LIN {X 0,Y 353.94,Z 241.157,A -85,B 0,C 180,E1 -13393.452,E2 -13393.452} C_VEL
LIN {X 0,Y 355.992,Z 254.031,A -85,B 0,C 180,E1 -13394.17,E2 -13394.17} C_VEL
LIN {X 0,Y 356.994,Z 264.311,A -85,B 0,C 180,E1 -13394.928,E2 -13394.928} C_VEL
LIN {X 0,Y 357.262,Z 272.08,A -85,B 0,C 180,E1 -13395.62,E2 -13395.62} C_VEL
LIN {X 0,Y 356.698,Z 280.213,A -85,B 0,C 180,E1 -13396.469,E2 -13396.469} C_VEL
LIN {X 0,Y 355.831,Z 287.972,A -85,B 0,C 180,E1 -13397.452,E2 -13397.452} C_VEL
LIN {X 0,Y 355.018,Z 296.94,A -85,B 0,C 180,E1 -13398.872,E2 -13398.872} C_VEL
LIN {X 0,Y 354.362,Z 303.882,A -85,B 0,C 180,E1 -13400.295,E2 -13400.295} C_VEL
LIN {X 0,Y 353.942,Z 308.46,A -85,B 0,C 180,E1 -13401.436,E2 -13401.436} C_VEL
LIN {X 0,Y 353.645,Z 312.278,A -85,B 0,C 180,E1 -13402.578,E2 -13402.578} C_VEL
LIN {X 0,Y 353.331,Z 316.635,A -85,B 0,C 180,E1 -13404.293,E2 -13404.293} C_VEL
LIN {X 0,Y 353.333,Z 318.872,A -85,B 0,C 180,E1 -13405.437,E2 -13405.437} C_VEL
LIN {X 0,Y 353.267,Z 320.538,A -85,B 0,C 180,E1 -13406.579,E2 -13406.579} C_VEL
LIN {X 0,Y 353.258,Z 321.597,A -85,B 0,C 180,E1 -13407.72,E2 -13407.72} C_VEL
LIN {X 0,Y 353.356,Z 322.159,A -85,B 0,C 180,E1 -13408.861,E2 -13408.861} C_VEL
LIN {X 0,Y 353.398,Z 322.239,A -85,B 0,C 180,E1 -13410,E2 -13410} C_VEL
LIN {X 0,Y 353.391,Z 321.836,A -85,B 0,C 180,E1 -13411.14,E2 -13411.14} C_VEL
LIN {X 0,Y 353.284,Z 320.881,A -85,B 0,C 180,E1 -13412.28,E2 -13412.28} C_VEL
LIN {X 0,Y 353.338,Z 318.39,A -85,B 0,C 180,E1 -13413.992,E2 -13413.992} C_VEL
LIN {X 0,Y 353.347,Z 316.056,A -85,B 0,C 180,E1 -13415.135,E2 -13415.135} C_VEL
LIN {X 0,Y 353.522,Z 311.248,A -85,B 0,C 180,E1 -13416.851,E2 -13416.851} C_VEL
LIN {X 0,Y 353.776,Z 306.025,A -85,B 0,C 180,E1 -13418.281,E2 -13418.281} C_VEL
LIN {X 0,Y 354.128,Z 300.895,A -85,B 0,C 180,E1 -13419.424,E2 -13419.424} C_VEL
LIN {X 0,Y 354.525,Z 294.697,A -85,B 0,C 180,E1 -13420.566,E2 -13420.566} C_VEL
LIN {X 0,Y 354.963,Z 288.171,A -85,B 0,C 180,E1 -13421.565,E2 -13421.565} C_VEL
LIN {X 0,Y 355.624,Z 280.281,A -85,B 0,C 180,E1 -13422.556,E2 -13422.556} C_VEL
LIN {X 0,Y 356.12,Z 271.928,A -85,B 0,C 180,E1 -13423.408,E2 -13423.408} C_VEL
LIN {X 0,Y 355.694,Z 262.322,A -85,B 0,C 180,E1 -13424.209,E2 -13424.209} C_VEL
LIN {X 0,Y 354.598,Z 250.562,A -85,B 0,C 180,E1 -13424.931,E2 -13424.931} C_VEL
LIN {X 0,Y 353.691,Z 242.124,A -85,B 0,C 180,E1 -13425.339,E2 -13425.339} C_VEL
LIN {X 0,Y 354.181,Z 233.988,A -85,B 0,C 180,E1 -13429.112,E2 -13429.112} C_VEL
LIN {X 0,Y 354.734,Z 226.313,A -85,B 0,C 180,E1 -13432.727,E2 -13432.727} C_VEL
LIN {X 0,Y 355.482,Z 218.591,A -85,B 0,C 180,E1 -13436.413,E2 -13436.413} C_VEL
LIN {X 0,Y 356.416,Z 210.762,A -85,B 0,C 180,E1 -13440.247,E2 -13440.247} C_VEL
LIN {X 0,Y 356.568,Z 207.213,A -85,B 0,C 180,E1 -13442.055,E2 -13442.055} C_VEL
LIN {X 0,Y 355.731,Z 201.801,A -85,B 0,C 180,E1 -13444.956,E2 -13444.956} C_VEL
LIN {X 0,Y 354.893,Z 197.094,A -85,B 0,C 180,E1 -13447.615,E2 -13447.615} C_VEL
LIN {X 0,Y 354.791,Z 197.102,A -85,B 0,C 180,E1 -13451.171,E2 -13451.171} C_VEL
LIN {X 0,Y 354.767,Z 197.108,A -85,B 0,C 180,E1 -13454.506,E2 -13454.506} C_VEL
LIN {X 0,Y 354.794,Z 197.101,A -85,B 0,C 180,E1 -13457.662,E2 -13457.662} C_VEL
LIN {X 0,Y 354.789,Z 197.103,A -85,B 0,C 180,E1 -13460.662,E2 -13460.662} C_VEL
LIN {X 0,Y 354.826,Z 197.101,A -85,B 0,C 180,E1 -13464.301,E2 -13464.301} C_VEL
LIN {X 0,Y 354.791,Z 197.103,A -85,B 0,C 180,E1 -13467.666,E2 -13467.666} C_VEL
LIN {X 0,Y 354.851,Z 197.096,A -85,B 0,C 180,E1 -13471.618,E2 -13471.618} C_VEL
LIN {X 0,Y 354.903,Z 197.09,A -85,B 0,C 180,E1 -13474.172,E2 -13474.172} C_VEL
LIN {X 0,Y 354.82,Z 197.102,A -85,B 0,C 180,E1 -13477.892,E2 -13477.892} C_VEL
LIN {X 0,Y 354.927,Z 197.088,A -85,B 0,C 180,E1 -13481.891,E2 -13481.891} C_VEL
LIN {X 0,Y 354.947,Z 197.083,A -85,B 0,C 180,E1 -13485.98,E2 -13485.98} C_VEL
LIN {X 0,Y 354.96,Z 197.083,A -85,B 0,C 180,E1 -13489.734,E2 -13489.734} C_VEL
LIN {X 0,Y 355.115,Z 197.065,A -85,B 0,C 180,E1 -13493.179,E2 -13493.179} C_VEL
LIN {X 0,Y 355.246,Z 197.046,A -85,B 0,C 180,E1 -13497.731,E2 -13497.731} C_VEL
LIN {X 0,Y 355.377,Z 197.028,A -85,B 0,C 180,E1 -13499.999,E2 -13499.999} C_VEL
LIN {X 0,Y 355.247,Z 197.044,A -85,B 0,C 180,E1 -13502.267,E2 -13502.267} C_VEL
LIN {X 0,Y 355.114,Z 197.065,A -85,B 0,C 180,E1 -13506.819,E2 -13506.819} C_VEL
LIN {X 0,Y 354.958,Z 197.081,A -85,B 0,C 180,E1 -13510.264,E2 -13510.264} C_VEL
LIN {X 0,Y 354.944,Z 197.082,A -85,B 0,C 180,E1 -13514.018,E2 -13514.018} C_VEL
LIN {X 0,Y 354.89,Z 197.089,A -85,B 0,C 180,E1 -13518.091,E2 -13518.091} C_VEL
LIN {X 0,Y 354.816,Z 197.1,A -85,B 0,C 180,E1 -13522.106,E2 -13522.106} C_VEL
LIN {X 0,Y 354.898,Z 197.088,A -85,B 0,C 180,E1 -13525.826,E2 -13525.826} C_VEL
LIN {X 0,Y 354.852,Z 197.094,A -85,B 0,C 180,E1 -13529.677,E2 -13529.677} C_VEL
LIN {X 0,Y 354.804,Z 197.101,A -85,B 0,C 180,E1 -13533.701,E2 -13533.701} C_VEL
LIN {X 0,Y 354.796,Z 197.104,A -85,B 0,C 180,E1 -13536.458,E2 -13536.458} C_VEL
LIN {X 0,Y 354.821,Z 197.097,A -85,B 0,C 180,E1 -13539.422,E2 -13539.422} C_VEL
LIN {X 0,Y 354.784,Z 197.102,A -85,B 0,C 180,E1 -13542.866,E2 -13542.866} C_VEL
LIN {X 0,Y 354.763,Z 197.108,A -85,B 0,C 180,E1 -13546.102,E2 -13546.102} C_VEL
LIN {X 0,Y 354.783,Z 197.103,A -85,B 0,C 180,E1 -13549.178,E2 -13549.178} C_VEL
LIN {X 0,Y 354.802,Z 197.1,A -85,B 0,C 180,E1 -13552.401,E2 -13552.401} C_VEL
LIN {X 0,Y 354.806,Z 197.099,A -85,B 0,C 180,E1 -13554.94,E2 -13554.94} C_VEL
LIN {X 0,Y 354.787,Z 197.102,A -85,B 0,C 180,E1 -13558.404,E2 -13558.404} C_VEL
LIN {X 0,Y 354.847,Z 197.098,A -85,B 0,C 180,E1 -13561.618,E2 -13561.618} C_VEL
LIN {X 0,Y 354.892,Z 197.089,A -85,B 0,C 180,E1 -13564.172,E2 -13564.172} C_VEL
LIN {X 0,Y 354.827,Z 197.098,A -85,B 0,C 180,E1 -13567.893,E2 -13567.893} C_VEL
LIN {X 0,Y 354.915,Z 197.086,A -85,B 0,C 180,E1 -13571.891,E2 -13571.891} C_VEL
LIN {X 0,Y 354.935,Z 197.083,A -85,B 0,C 180,E1 -13575.98,E2 -13575.98} C_VEL
LIN {X 0,Y 354.975,Z 197.078,A -85,B 0,C 180,E1 -13579.736,E2 -13579.736} C_VEL
LIN {X 0,Y 355.105,Z 197.062,A -85,B 0,C 180,E1 -13582.036,E2 -13582.036} C_VEL
LIN {X 0,Y 355.084,Z 197.065,A -85,B 0,C 180,E1 -13584.32,E2 -13584.32} C_VEL
LIN {X 0,Y 355.235,Z 197.045,A -85,B 0,C 180,E1 -13587.732,E2 -13587.732} C_VEL
LIN {X 0,Y 355.388,Z 197.027,A -85,B 0,C 180,E1 -13590,E2 -13590} C_VEL
LIN {X 0,Y 355.237,Z 197.047,A -85,B 0,C 180,E1 -13592.267,E2 -13592.267} C_VEL
LIN {X 0,Y 355.131,Z 197.062,A -85,B 0,C 180,E1 -13596.819,E2 -13596.819} C_VEL
LIN {X 0,Y 355.001,Z 197.076,A -85,B 0,C 180,E1 -13599.113,E2 -13599.113} C_VEL
LIN {X 0,Y 354.834,Z 197.1,A -85,B 0,C 180,E1 -13602.584,E2 -13602.584} C_VEL
LIN {X 0,Y 354.529,Z 197.156,A -85,B 0,C 180,E1 -13605.375,E2 -13605.375} C_VEL
LIN {X 0,Y 354.19,Z 201.044,A -85,B 0,C 180,E1 -13608.51,E2 -13608.51} C_VEL
LIN {X 0,Y 353.974,Z 205.678,A -85,B 0,C 180,E1 -13612.162,E2 -13612.162} C_VEL
LIN {X 0,Y 353.844,Z 208.876,A -85,B 0,C 180,E1 -13614.651,E2 -13614.651} C_VEL
LIN {X 0,Y 353.691,Z 212.209,A -85,B 0,C 180,E1 -13617.195,E2 -13617.195} C_VEL
LIN {X 0,Y 353.563,Z 216.799,A -85,B 0,C 180,E1 -13620.663,E2 -13620.663} C_VEL
LIN {X 0,Y 355.402,Z 227.901,A -85,B 0,C 180,E1 -13621.298,E2 -13621.298} C_VEL
LIN {X 0,Y 356.573,Z 235.778,A -85,B 0,C 180,E1 -13621.886,E2 -13621.886} C_VEL
LIN {X 0,Y 356.726,Z 240.779,A -85,B 0,C 180,E1 -13622.303,E2 -13622.303} C_VEL
LIN {X 0,Y 356.17,Z 249.655,A -85,B 0,C 180,E1 -13623.2,E2 -13623.2} C_VEL
LIN {X 0,Y 355.669,Z 257.094,A -85,B 0,C 180,E1 -13624.132,E2 -13624.132} C_VEL
LIN {X 0,Y 355.113,Z 264.014,A -85,B 0,C 180,E1 -13625.189,E2 -13625.189} C_VEL
LIN {X 0,Y 354.591,Z 270.903,A -85,B 0,C 180,E1 -13626.484,E2 -13626.484} C_VEL
LIN {X 0,Y 354.16,Z 277.029,A -85,B 0,C 180,E1 -13627.964,E2 -13627.964} C_VEL
LIN {X 0,Y 353.727,Z 281.835,A -85,B 0,C 180,E1 -13629.478,E2 -13629.478} C_VEL
LIN {X 0,Y 353.468,Z 285.305,A -85,B 0,C 180,E1 -13630.929,E2 -13630.929} C_VEL
LIN {X 0,Y 353.266,Z 288.109,A -85,B 0,C 180,E1 -13632.603,E2 -13632.603} C_VEL
LIN {X 0,Y 353.172,Z 289.652,A -85,B 0,C 180,E1 -13634.245,E2 -13634.245} C_VEL
LIN {X 0,Y 353.191,Z 290.008,A -85,B 0,C 180,E1 -13635.859,E2 -13635.859} C_VEL
LIN {X 0,Y 353.335,Z 289.319,A -85,B 0,C 180,E1 -13637.449,E2 -13637.449} C_VEL
LIN {X 0,Y 353.635,Z 287.419,A -85,B 0,C 180,E1 -13639.15,E2 -13639.15} C_VEL
LIN {X 0,Y 353.136,Z 285.956,A -85,B 0,C 180,E1 -13640.076,E2 -13640.076} C_VEL
LIN {X 0,Y 350.647,Z 283.004,A -85,B 0,C 180,E1 -13641.571,E2 -13641.571} C_VEL
LIN {X 0,Y 348.304,Z 279.171,A -85,B 0,C 180,E1 -13643.022,E2 -13643.022} C_VEL
LIN {X 0,Y 348.029,Z 276.23,A -85,B 0,C 180,E1 -13643.864,E2 -13643.864} C_VEL
LIN {X 0,Y 348.715,Z 270.077,A -85,B 0,C 180,E1 -13645.297,E2 -13645.297} C_VEL
LIN {X 0,Y 349.518,Z 263.05,A -85,B 0,C 180,E1 -13646.604,E2 -13646.604} C_VEL
LIN {X 0,Y 350.516,Z 254.114,A -85,B 0,C 180,E1 -13647.906,E2 -13647.906} C_VEL
LIN {X 0,Y 351.121,Z 246.314,A -85,B 0,C 180,E1 -13648.805,E2 -13648.805} C_VEL
LIN {X 0,Y 351.522,Z 241.461,A -85,B 0,C 180,E1 -13649.283,E2 -13649.283} C_VEL
LIN {X 0,Y 350.018,Z 231.844,A -85,B 0,C 180,E1 -13650.158,E2 -13650.158} C_VEL
LIN {X 0,Y 347.72,Z 221.982,A -85,B 0,C 180,E1 -13650.895,E2 -13650.895} C_VEL
LIN {X 0,Y 346.82,Z 218.272,A -85,B 0,C 180,E1 -13651.15,E2 -13651.15} C_VEL
LIN {X 0,Y 346.982,Z 215.406,A -85,B 0,C 180,E1 -13653.54,E2 -13653.54} C_VEL
LIN {X 0,Y 347.236,Z 210.883,A -85,B 0,C 180,E1 -13657.385,E2 -13657.385} C_VEL
LIN {X 0,Y 347.542,Z 206.631,A -85,B 0,C 180,E1 -13661.123,E2 -13661.123} C_VEL
LIN {X 0,Y 347.864,Z 202.634,A -85,B 0,C 180,E1 -13664.774,E2 -13664.774} C_VEL
LIN {X 0,Y 347.994,Z 200.093,A -85,B 0,C 180,E1 -13667.166,E2 -13667.166} C_VEL
LIN {X 0,Y 347.885,Z 197.966,A -85,B 0,C 180,E1 -13669.525,E2 -13669.525} C_VEL
LIN {X 0,Y 348.079,Z 197.946,A -85,B 0,C 180,E1 -13671.876,E2 -13671.876} C_VEL
LIN {X 0,Y 348.068,Z 197.949,A -85,B 0,C 180,E1 -13674.207,E2 -13674.207} C_VEL
LIN {X 0,Y 348.207,Z 197.926,A -85,B 0,C 180,E1 -13677.688,E2 -13677.688} C_VEL
LIN {X 0,Y 348.369,Z 197.905,A -85,B 0,C 180,E1 -13680.001,E2 -13680.001} C_VEL
LIN {X 0,Y 348.207,Z 197.926,A -85,B 0,C 180,E1 -13682.314,E2 -13682.314} C_VEL
LIN {X 0,Y 348.081,Z 197.942,A -85,B 0,C 180,E1 -13686.959,E2 -13686.959} C_VEL
LIN {X 0,Y 347.899,Z 197.963,A -85,B 0,C 180,E1 -13690.476,E2 -13690.476} C_VEL
LIN {X 0,Y 347.9,Z 197.963,A -85,B 0,C 180,E1 -13694.151,E2 -13694.151} C_VEL
LIN {X 0,Y 347.894,Z 197.964,A -85,B 0,C 180,E1 -13698.291,E2 -13698.291} C_VEL
LIN {X 0,Y 347.791,Z 197.977,A -85,B 0,C 180,E1 -13701.636,E2 -13701.636} C_VEL
LIN {X 0,Y 347.814,Z 197.97,A -85,B 0,C 180,E1 -13705.109,E2 -13705.109} C_VEL
LIN {X 0,Y 347.812,Z 197.974,A -85,B 0,C 180,E1 -13707.695,E2 -13707.695} C_VEL
LIN {X 0,Y 347.766,Z 197.979,A -85,B 0,C 180,E1 -13710.347,E2 -13710.347} C_VEL
LIN {X 0,Y 347.746,Z 197.982,A -85,B 0,C 180,E1 -13714.464,E2 -13714.464} C_VEL
LIN {X 0,Y 347.775,Z 197.98,A -85,B 0,C 180,E1 -13717.989,E2 -13717.989} C_VEL
LIN {X 0,Y 347.753,Z 197.984,A -85,B 0,C 180,E1 -13721.831,E2 -13721.831} C_VEL
LIN {X 0,Y 347.708,Z 197.991,A -85,B 0,C 180,E1 -13725.027,E2 -13725.027} C_VEL
LIN {X 0,Y 347.79,Z 198.146,A -85,B 0,C 180,E1 -13728.948,E2 -13728.948} C_VEL
LIN {X 0,Y 348.556,Z 202.078,A -85,B 0,C 180,E1 -13731.848,E2 -13731.848} C_VEL
LIN {X 0,Y 349.657,Z 207.924,A -85,B 0,C 180,E1 -13735.751,E2 -13735.751} C_VEL
LIN {X 0,Y 350.09,Z 210.716,A -85,B 0,C 180,E1 -13737.475,E2 -13737.475} C_VEL
LIN {X 0,Y 349.935,Z 213.693,A -85,B 0,C 180,E1 -13739.195,E2 -13739.195} C_VEL
LIN {X 0,Y 348.847,Z 220.858,A -85,B 0,C 180,E1 -13743.045,E2 -13743.045} C_VEL
LIN {X 0,Y 347.96,Z 228.169,A -85,B 0,C 180,E1 -13746.806,E2 -13746.806} C_VEL
LIN {X 0,Y 347.292,Z 235.615,A -85,B 0,C 180,E1 -13750.494,E2 -13750.494} C_VEL
LIN {X 0,Y 346.929,Z 241.06,A -85,B 0,C 180,E1 -13753.051,E2 -13753.051} C_VEL
LIN {X 0,Y 349.037,Z 253.685,A -85,B 0,C 180,E1 -13753.777,E2 -13753.777} C_VEL
LIN {X 0,Y 350.037,Z 263.552,A -85,B 0,C 180,E1 -13754.525,E2 -13754.525} C_VEL
LIN {X 0,Y 350.341,Z 272.338,A -85,B 0,C 180,E1 -13755.329,E2 -13755.329} C_VEL
LIN {X 0,Y 349.815,Z 280.367,A -85,B 0,C 180,E1 -13756.198,E2 -13756.198} C_VEL
LIN {X 0,Y 348.917,Z 288.047,A -85,B 0,C 180,E1 -13757.199,E2 -13757.199} C_VEL
LIN {X 0,Y 348.057,Z 296.92,A -85,B 0,C 180,E1 -13758.646,E2 -13758.646} C_VEL
LIN {X 0,Y 347.339,Z 303.789,A -85,B 0,C 180,E1 -13760.097,E2 -13760.097} C_VEL
LIN {X 0,Y 346.903,Z 308.325,A -85,B 0,C 180,E1 -13761.261,E2 -13761.261} C_VEL
LIN {X 0,Y 346.572,Z 312.11,A -85,B 0,C 180,E1 -13762.426,E2 -13762.426} C_VEL
LIN {X 0,Y 346.251,Z 316.425,A -85,B 0,C 180,E1 -13764.175,E2 -13764.175} C_VEL
LIN {X 0,Y 346.245,Z 318.624,A -85,B 0,C 180,E1 -13765.343,E2 -13765.343} C_VEL
LIN {X 0,Y 346.189,Z 320.273,A -85,B 0,C 180,E1 -13766.509,E2 -13766.509} C_VEL
LIN {X 0,Y 346.164,Z 321.315,A -85,B 0,C 180,E1 -13767.673,E2 -13767.673} C_VEL
LIN {X 0,Y 346.257,Z 321.845,A -85,B 0,C 180,E1 -13768.837,E2 -13768.837} C_VEL
LIN {X 0,Y 346.318,Z 321.895,A -85,B 0,C 180,E1 -13770,E2 -13770} C_VEL
LIN {X 0,Y 346.294,Z 321.46,A -85,B 0,C 180,E1 -13771.163,E2 -13771.163} C_VEL
LIN {X 0,Y 346.188,Z 320.496,A -85,B 0,C 180,E1 -13772.327,E2 -13772.327} C_VEL
LIN {X 0,Y 346.269,Z 317.952,A -85,B 0,C 180,E1 -13774.074,E2 -13774.074} C_VEL
LIN {X 0,Y 346.246,Z 315.595,A -85,B 0,C 180,E1 -13775.241,E2 -13775.241} C_VEL
LIN {X 0,Y 346.444,Z 310.731,A -85,B 0,C 180,E1 -13776.991,E2 -13776.991} C_VEL
LIN {X 0,Y 346.741,Z 305.465,A -85,B 0,C 180,E1 -13778.45,E2 -13778.45} C_VEL
LIN {X 0,Y 347.065,Z 300.279,A -85,B 0,C 180,E1 -13779.617,E2 -13779.617} C_VEL
LIN {X 0,Y 347.534,Z 294.026,A -85,B 0,C 180,E1 -13780.781,E2 -13780.781} C_VEL
LIN {X 0,Y 348.111,Z 286.412,A -85,B 0,C 180,E1 -13781.943,E2 -13781.943} C_VEL
LIN {X 0,Y 348.889,Z 276.928,A -85,B 0,C 180,E1 -13783.098,E2 -13783.098} C_VEL
LIN {X 0,Y 349.088,Z 269.405,A -85,B 0,C 180,E1 -13783.832,E2 -13783.832} C_VEL
LIN {X 0,Y 348.361,Z 259.219,A -85,B 0,C 180,E1 -13784.63,E2 -13784.63} C_VEL
LIN {X 0,Y 347.423,Z 249.351,A -85,B 0,C 180,E1 -13785.218,E2 -13785.218} C_VEL
LIN {X 0,Y 346.638,Z 241.909,A -85,B 0,C 180,E1 -13785.584,E2 -13785.584} C_VEL
LIN {X 0,Y 347.139,Z 233.624,A -85,B 0,C 180,E1 -13789.515,E2 -13789.515} C_VEL
LIN {X 0,Y 347.646,Z 227.22,A -85,B 0,C 180,E1 -13792.588,E2 -13792.588} C_VEL
LIN {X 0,Y 348.397,Z 219.537,A -85,B 0,C 180,E1 -13796.346,E2 -13796.346} C_VEL
LIN {X 0,Y 349.352,Z 211.86,A -85,B 0,C 180,E1 -13800.194,E2 -13800.194} C_VEL
LIN {X 0,Y 349.616,Z 209.278,A -85,B 0,C 180,E1 -13801.511,E2 -13801.511} C_VEL
LIN {X 0,Y 348.935,Z 204.077,A -85,B 0,C 180,E1 -13804.33,E2 -13804.33} C_VEL
LIN {X 0,Y 347.841,Z 197.972,A -85,B 0,C 180,E1 -13807.899,E2 -13807.899} C_VEL
LIN {X 0,Y 347.754,Z 197.978,A -85,B 0,C 180,E1 -13811.83,E2 -13811.83} C_VEL
LIN {X 0,Y 347.709,Z 197.984,A -85,B 0,C 180,E1 -13815.027,E2 -13815.027} C_VEL
LIN {X 0,Y 347.751,Z 197.982,A -85,B 0,C 180,E1 -13818.398,E2 -13818.398} C_VEL
LIN {X 0,Y 347.768,Z 197.979,A -85,B 0,C 180,E1 -13822.013,E2 -13822.013} C_VEL
LIN {X 0,Y 347.749,Z 197.979,A -85,B 0,C 180,E1 -13825.536,E2 -13825.536} C_VEL
LIN {X 0,Y 347.749,Z 197.981,A -85,B 0,C 180,E1 -13828.3,E2 -13828.3} C_VEL
LIN {X 0,Y 347.783,Z 197.974,A -85,B 0,C 180,E1 -13830.987,E2 -13830.987} C_VEL
LIN {X 0,Y 347.835,Z 197.97,A -85,B 0,C 180,E1 -13833.607,E2 -13833.607} C_VEL
LIN {X 0,Y 347.789,Z 197.976,A -85,B 0,C 180,E1 -13836.161,E2 -13836.161} C_VEL
LIN {X 0,Y 347.813,Z 197.974,A -85,B 0,C 180,E1 -13839.909,E2 -13839.909} C_VEL
LIN {X 0,Y 347.871,Z 197.963,A -85,B 0,C 180,E1 -13842.359,E2 -13842.359} C_VEL
LIN {X 0,Y 347.902,Z 197.961,A -85,B 0,C 180,E1 -13845.97,E2 -13845.97} C_VEL
LIN {X 0,Y 347.901,Z 197.964,A -85,B 0,C 180,E1 -13849.524,E2 -13849.524} C_VEL
LIN {X 0,Y 348.081,Z 197.939,A -85,B 0,C 180,E1 -13853.041,E2 -13853.041} C_VEL
LIN {X 0,Y 348.209,Z 197.922,A -85,B 0,C 180,E1 -13857.686,E2 -13857.686} C_VEL
LIN {X 0,Y 348.327,Z 197.906,A -85,B 0,C 180,E1 -13859.999,E2 -13859.999} C_VEL
LIN {X 0,Y 348.209,Z 197.921,A -85,B 0,C 180,E1 -13862.312,E2 -13862.312} C_VEL
LIN {X 0,Y 348.08,Z 197.942,A -85,B 0,C 180,E1 -13866.957,E2 -13866.957} C_VEL
LIN {X 0,Y 347.899,Z 197.961,A -85,B 0,C 180,E1 -13870.474,E2 -13870.474} C_VEL
LIN {X 0,Y 347.9,Z 197.96,A -85,B 0,C 180,E1 -13874.149,E2 -13874.149} C_VEL
LIN {X 0,Y 347.829,Z 197.97,A -85,B 0,C 180,E1 -13878.258,E2 -13878.258} C_VEL
LIN {X 0,Y 347.767,Z 197.976,A -85,B 0,C 180,E1 -13881.625,E2 -13881.625} C_VEL
LIN {X 0,Y 347.81,Z 197.971,A -85,B 0,C 180,E1 -13885.107,E2 -13885.107} C_VEL
LIN {X 0,Y 347.81,Z 197.971,A -85,B 0,C 180,E1 -13887.692,E2 -13887.692} C_VEL
LIN {X 0,Y 347.762,Z 197.981,A -85,B 0,C 180,E1 -13890.345,E2 -13890.345} C_VEL
LIN {X 0,Y 347.742,Z 197.982,A -85,B 0,C 180,E1 -13894.463,E2 -13894.463} C_VEL
LIN {X 0,Y 347.771,Z 197.98,A -85,B 0,C 180,E1 -13897.987,E2 -13897.987} C_VEL
LIN {X 0,Y 347.747,Z 197.982,A -85,B 0,C 180,E1 -13901.829,E2 -13901.829} C_VEL
LIN {X 0,Y 347.701,Z 197.984,A -85,B 0,C 180,E1 -13905.026,E2 -13905.026} C_VEL
LIN {X 0,Y 347.745,Z 197.98,A -85,B 0,C 180,E1 -13908.396,E2 -13908.396} C_VEL
LIN {X 0,Y 347.769,Z 197.979,A -85,B 0,C 180,E1 -13912.01,E2 -13912.01} C_VEL
LIN {X 0,Y 347.738,Z 197.984,A -85,B 0,C 180,E1 -13915.535,E2 -13915.535} C_VEL
LIN {X 0,Y 347.758,Z 197.982,A -85,B 0,C 180,E1 -13919.653,E2 -13919.653} C_VEL
LIN {X 0,Y 347.846,Z 197.966,A -85,B 0,C 180,E1 -13922.743,E2 -13922.743} C_VEL
LIN {X 0,Y 347.781,Z 197.974,A -85,B 0,C 180,E1 -13926.161,E2 -13926.161} C_VEL
LIN {X 0,Y 347.81,Z 197.971,A -85,B 0,C 180,E1 -13929.909,E2 -13929.909} C_VEL
LIN {X 0,Y 347.859,Z 197.964,A -85,B 0,C 180,E1 -13932.359,E2 -13932.359} C_VEL
LIN {X 0,Y 347.889,Z 197.96,A -85,B 0,C 180,E1 -13935.97,E2 -13935.97} C_VEL
LIN {X 0,Y 347.925,Z 197.957,A -85,B 0,C 180,E1 -13939.525,E2 -13939.525} C_VEL
LIN {X 0,Y 348.066,Z 197.939,A -85,B 0,C 180,E1 -13941.874,E2 -13941.874} C_VEL
LIN {X 0,Y 348.059,Z 197.94,A -85,B 0,C 180,E1 -13944.205,E2 -13944.205} C_VEL
LIN {X 0,Y 348.197,Z 197.922,A -85,B 0,C 180,E1 -13947.686,E2 -13947.686} C_VEL
LIN {X 0,Y 348.337,Z 197.905,A -85,B 0,C 180,E1 -13950,E2 -13950} C_VEL
LIN {X 0,Y 348.199,Z 197.924,A -85,B 0,C 180,E1 -13952.313,E2 -13952.313} C_VEL
LIN {X 0,Y 348.099,Z 197.937,A -85,B 0,C 180,E1 -13956.958,E2 -13956.958} C_VEL
LIN {X 0,Y 347.936,Z 197.955,A -85,B 0,C 180,E1 -13959.299,E2 -13959.299} C_VEL
LIN {X 0,Y 347.79,Z 197.975,A -85,B 0,C 180,E1 -13962.843,E2 -13962.843} C_VEL
LIN {X 0,Y 347.442,Z 198.211,A -85,B 0,C 180,E1 -13965.546,E2 -13965.546} C_VEL
LIN {X 0,Y 347.112,Z 202.33,A -85,B 0,C 180,E1 -13968.902,E2 -13968.902} C_VEL
LIN {X 0,Y 346.975,Z 205.423,A -85,B 0,C 180,E1 -13971.382,E2 -13971.382} C_VEL
LIN {X 0,Y 346.746,Z 210.268,A -85,B 0,C 180,E1 -13975.191,E2 -13975.191} C_VEL
LIN {X 0,Y 346.575,Z 213.619,A -85,B 0,C 180,E1 -13977.801,E2 -13977.801} C_VEL
LIN {X 0,Y 346.505,Z 217.067,A -85,B 0,C 180,E1 -13980.424,E2 -13980.424} C_VEL
LIN {X 0,Y 348.301,Z 227.835,A -85,B 0,C 180,E1 -13981.051,E2 -13981.051} C_VEL
LIN {X 0,Y 349.549,Z 236.356,A -85,B 0,C 180,E1 -13981.7,E2 -13981.7} C_VEL
LIN {X 0,Y 349.73,Z 241.206,A -85,B 0,C 180,E1 -13982.116,E2 -13982.116} C_VEL
LIN {X 0,Y 349.122,Z 250.603,A -85,B 0,C 180,E1 -13983.096,E2 -13983.096} C_VEL
LIN {X 0,Y 348.578,Z 258.652,A -85,B 0,C 180,E1 -13984.148,E2 -13984.148} C_VEL
LIN {X 0,Y 347.867,Z 266.954,A -85,B 0,C 180,E1 -13985.509,E2 -13985.509} C_VEL
LIN {X 0,Y 347.357,Z 273.993,A -85,B 0,C 180,E1 -13987.023,E2 -13987.023} C_VEL
LIN {X 0,Y 346.934,Z 278.896,A -85,B 0,C 180,E1 -13988.344,E2 -13988.344} C_VEL
LIN {X 0,Y 346.599,Z 282.619,A -85,B 0,C 180,E1 -13989.601,E2 -13989.601} C_VEL
LIN {X 0,Y 346.326,Z 286.508,A -85,B 0,C 180,E1 -13991.339,E2 -13991.339} C_VEL
LIN {X 0,Y 346.13,Z 288.929,A -85,B 0,C 180,E1 -13993.035,E2 -13993.035} C_VEL
LIN {X 0,Y 346.066,Z 290.317,A -85,B 0,C 180,E1 -13995.299,E2 -13995.299} C_VEL
LIN {X 0,Y 346.177,Z 290.088,A -85,B 0,C 180,E1 -13996.959,E2 -13996.959} C_VEL
LIN {X 0,Y 346.452,Z 288.663,A -85,B 0,C 180,E1 -13998.64,E2 -13998.64} C_VEL
LIN {X 0,Y 346.806,Z 285.979,A -85,B 0,C 180,E1 -14000.36,E2 -14000.36} C_VEL
LIN {X 0,Y 347.161,Z 283.128,A -85,B 0,C 180,E1 -14001.648,E2 -14001.648} C_VEL
LIN {X 0,Y 347.788,Z 278.206,A -85,B 0,C 180,E1 -14003.315,E2 -14003.315} C_VEL
LIN {X 0,Y 348.029,Z 276.23,A -85,B 0,C 180,E1 -14003.864,E2 -14003.864} C_VEL
LIN {X 0,Y 347.773,Z 273.111,A -85,B 0,C 180,E1 -14004.676,E2 -14004.676} C_VEL
LIN {X 0,Y 345.608,Z 267.605,A -85,B 0,C 180,E1 -14005.986,E2 -14005.986} C_VEL
LIN {X 0,Y 343.539,Z 261.333,A -85,B 0,C 180,E1 -14007.228,E2 -14007.228} C_VEL
LIN {X 0,Y 343.409,Z 256.965,A -85,B 0,C 180,E1 -14007.905,E2 -14007.905} C_VEL
LIN {X 0,Y 344.348,Z 246.796,A -85,B 0,C 180,E1 -14009.147,E2 -14009.147} C_VEL
LIN {X 0,Y 344.711,Z 242.533,A -85,B 0,C 180,E1 -14009.578,E2 -14009.578} C_VEL
LIN {X 0,Y 343.087,Z 232.251,A -85,B 0,C 180,E1 -14010.554,E2 -14010.554} C_VEL
LIN {X 0,Y 340.653,Z 222.105,A -85,B 0,C 180,E1 -14011.338,E2 -14011.338} C_VEL
LIN {X 0,Y 339.8,Z 218.575,A -85,B 0,C 180,E1 -14011.596,E2 -14011.596} C_VEL
LIN {X 0,Y 340.036,Z 213.92,A -85,B 0,C 180,E1 -14015.585,E2 -14015.585} C_VEL
LIN {X 0,Y 340.354,Z 209.546,A -85,B 0,C 180,E1 -14019.451,E2 -14019.451} C_VEL
LIN {X 0,Y 340.648,Z 206.74,A -85,B 0,C 180,E1 -14021.974,E2 -14021.974} C_VEL
LIN {X 0,Y 340.949,Z 202.812,A -85,B 0,C 180,E1 -14025.68,E2 -14025.68} C_VEL
LIN {X 0,Y 340.955,Z 200.362,A -85,B 0,C 180,E1 -14028.106,E2 -14028.106} C_VEL
LIN {X 0,Y 340.893,Z 199.19,A -85,B 0,C 180,E1 -14029.308,E2 -14029.308} C_VEL
LIN {X 0,Y 341.043,Z 198.822,A -85,B 0,C 180,E1 -14031.707,E2 -14031.707} C_VEL
LIN {X 0,Y 341.044,Z 198.825,A -85,B 0,C 180,E1 -14034.087,E2 -14034.087} C_VEL
LIN {X 0,Y 341.169,Z 198.803,A -85,B 0,C 180,E1 -14037.64,E2 -14037.64} C_VEL
LIN {X 0,Y 341.317,Z 198.783,A -85,B 0,C 180,E1 -14040.001,E2 -14040.001} C_VEL
LIN {X 0,Y 341.169,Z 198.803,A -85,B 0,C 180,E1 -14042.362,E2 -14042.362} C_VEL
LIN {X 0,Y 341.049,Z 198.817,A -85,B 0,C 180,E1 -14047.103,E2 -14047.103} C_VEL
LIN {X 0,Y 340.85,Z 198.842,A -85,B 0,C 180,E1 -14050.695,E2 -14050.695} C_VEL
LIN {X 0,Y 340.865,Z 198.838,A -85,B 0,C 180,E1 -14054.326,E2 -14054.326} C_VEL
LIN {X 0,Y 340.84,Z 198.843,A -85,B 0,C 180,E1 -14058.468,E2 -14058.468} C_VEL
LIN {X 0,Y 340.756,Z 198.853,A -85,B 0,C 180,E1 -14061.858,E2 -14061.858} C_VEL
LIN {X 0,Y 340.775,Z 198.846,A -85,B 0,C 180,E1 -14065.665,E2 -14065.665} C_VEL
LIN {X 0,Y 340.742,Z 198.855,A -85,B 0,C 180,E1 -14068.32,E2 -14068.32} C_VEL
LIN {X 0,Y 340.706,Z 198.859,A -85,B 0,C 180,E1 -14071.045,E2 -14071.045} C_VEL
LIN {X 0,Y 340.72,Z 198.856,A -85,B 0,C 180,E1 -14075.279,E2 -14075.279} C_VEL
LIN {X 0,Y 340.712,Z 198.859,A -85,B 0,C 180,E1 -14078.386,E2 -14078.386} C_VEL
LIN {X 0,Y 340.701,Z 198.863,A -85,B 0,C 180,E1 -14082.046,E2 -14082.046} C_VEL
LIN {X 0,Y 340.654,Z 198.869,A -85,B 0,C 180,E1 -14086.227,E2 -14086.227} C_VEL
LIN {X 0,Y 340.731,Z 198.987,A -85,B 0,C 180,E1 -14088.329,E2 -14088.329} C_VEL
LIN {X 0,Y 341.634,Z 203.675,A -85,B 0,C 180,E1 -14091.892,E2 -14091.892} C_VEL
LIN {X 0,Y 342.507,Z 208.437,A -85,B 0,C 180,E1 -14095.163,E2 -14095.163} C_VEL
LIN {X 0,Y 343.103,Z 212.604,A -85,B 0,C 180,E1 -14097.821,E2 -14097.821} C_VEL
LIN {X 0,Y 342.859,Z 215.359,A -85,B 0,C 180,E1 -14099.422,E2 -14099.422} C_VEL
LIN {X 0,Y 341.787,Z 222.053,A -85,B 0,C 180,E1 -14103.104,E2 -14103.104} C_VEL
LIN {X 0,Y 341.01,Z 228.107,A -85,B 0,C 180,E1 -14106.304,E2 -14106.304} C_VEL
LIN {X 0,Y 340.285,Z 235.513,A -85,B 0,C 180,E1 -14110.076,E2 -14110.076} C_VEL
LIN {X 0,Y 339.917,Z 240.583,A -85,B 0,C 180,E1 -14112.594,E2 -14112.594} C_VEL
LIN {X 0,Y 342.074,Z 253.386,A -85,B 0,C 180,E1 -14113.361,E2 -14113.361} C_VEL
LIN {X 0,Y 343.094,Z 263.082,A -85,B 0,C 180,E1 -14114.115,E2 -14114.115} C_VEL
LIN {X 0,Y 343.444,Z 271.242,A -85,B 0,C 180,E1 -14114.876,E2 -14114.876} C_VEL
LIN {X 0,Y 343.07,Z 279.368,A -85,B 0,C 180,E1 -14115.769,E2 -14115.769} C_VEL
LIN {X 0,Y 342.154,Z 287.139,A -85,B 0,C 180,E1 -14116.791,E2 -14116.791} C_VEL
LIN {X 0,Y 341.464,Z 293.586,A -85,B 0,C 180,E1 -14117.821,E2 -14117.821} C_VEL
LIN {X 0,Y 340.751,Z 299.75,A -85,B 0,C 180,E1 -14119.002,E2 -14119.002} C_VEL
LIN {X 0,Y 340.081,Z 306.072,A -85,B 0,C 180,E1 -14120.484,E2 -14120.484} C_VEL
LIN {X 0,Y 339.527,Z 311.937,A -85,B 0,C 180,E1 -14122.268,E2 -14122.268} C_VEL
LIN {X 0,Y 339.256,Z 315.007,A -85,B 0,C 180,E1 -14123.458,E2 -14123.458} C_VEL
LIN {X 0,Y 339.139,Z 318.378,A -85,B 0,C 180,E1 -14125.245,E2 -14125.245} C_VEL
LIN {X 0,Y 339.114,Z 320.008,A -85,B 0,C 180,E1 -14126.436,E2 -14126.436} C_VEL
LIN {X 0,Y 339.074,Z 321.038,A -85,B 0,C 180,E1 -14127.624,E2 -14127.624} C_VEL
LIN {X 0,Y 339.159,Z 321.532,A -85,B 0,C 180,E1 -14128.813,E2 -14128.813} C_VEL
LIN {X 0,Y 339.226,Z 321.546,A -85,B 0,C 180,E1 -14130,E2 -14130} C_VEL
LIN {X 0,Y 339.197,Z 321.074,A -85,B 0,C 180,E1 -14131.187,E2 -14131.187} C_VEL
LIN {X 0,Y 339.097,Z 320.09,A -85,B 0,C 180,E1 -14132.376,E2 -14132.376} C_VEL
LIN {X 0,Y 339.2,Z 317.488,A -85,B 0,C 180,E1 -14134.159,E2 -14134.159} C_VEL
LIN {X 0,Y 339.209,Z 313.422,A -85,B 0,C 180,E1 -14136.007,E2 -14136.007} C_VEL
LIN {X 0,Y 339.506,Z 308.253,A -85,B 0,C 180,E1 -14137.733,E2 -14137.733} C_VEL
LIN {X 0,Y 339.96,Z 301.029,A -85,B 0,C 180,E1 -14139.52,E2 -14139.52} C_VEL
LIN {X 0,Y 340.402,Z 294.985,A -85,B 0,C 180,E1 -14140.709,E2 -14140.709} C_VEL
LIN {X 0,Y 340.92,Z 287.614,A -85,B 0,C 180,E1 -14141.897,E2 -14141.897} C_VEL
LIN {X 0,Y 341.632,Z 279.739,A -85,B 0,C 180,E1 -14142.928,E2 -14142.928} C_VEL
LIN {X 0,Y 342.107,Z 271.393,A -85,B 0,C 180,E1 -14143.817,E2 -14143.817} C_VEL
LIN {X 0,Y 341.503,Z 261.169,A -85,B 0,C 180,E1 -14144.704,E2 -14144.704} C_VEL
LIN {X 0,Y 340.406,Z 249.59,A -85,B 0,C 180,E1 -14145.432,E2 -14145.432} C_VEL
LIN {X 0,Y 339.577,Z 241.639,A -85,B 0,C 180,E1 -14145.839,E2 -14145.839} C_VEL
LIN {X 0,Y 340.024,Z 234.507,A -85,B 0,C 180,E1 -14149.312,E2 -14149.312} C_VEL
LIN {X 0,Y 340.646,Z 226.868,A -85,B 0,C 180,E1 -14153.079,E2 -14153.079} C_VEL
LIN {X 0,Y 341.469,Z 219.201,A -85,B 0,C 180,E1 -14156.924,E2 -14156.924} C_VEL
LIN {X 0,Y 342.474,Z 211.518,A -85,B 0,C 180,E1 -14160.866,E2 -14160.866} C_VEL
LIN {X 0,Y 342.392,Z 208.123,A -85,B 0,C 180,E1 -14162.693,E2 -14162.693} C_VEL
LIN {X 0,Y 341.417,Z 202.537,A -85,B 0,C 180,E1 -14165.857,E2 -14165.857} C_VEL
LIN {X 0,Y 340.791,Z 198.85,A -85,B 0,C 180,E1 -14168.032,E2 -14168.032} C_VEL
LIN {X 0,Y 340.703,Z 198.857,A -85,B 0,C 180,E1 -14172.045,E2 -14172.045} C_VEL
LIN {X 0,Y 340.655,Z 198.866,A -85,B 0,C 180,E1 -14176.227,E2 -14176.227} C_VEL
LIN {X 0,Y 340.678,Z 198.86,A -85,B 0,C 180,E1 -14179.756,E2 -14179.756} C_VEL
LIN {X 0,Y 340.707,Z 198.855,A -85,B 0,C 180,E1 -14183.258,E2 -14183.258} C_VEL
LIN {X 0,Y 340.697,Z 198.861,A -85,B 0,C 180,E1 -14186.153,E2 -14186.153} C_VEL
LIN {X 0,Y 340.746,Z 198.853,A -85,B 0,C 180,E1 -14190.329,E2 -14190.329} C_VEL
LIN {X 0,Y 340.808,Z 198.842,A -85,B 0,C 180,E1 -14193.019,E2 -14193.019} C_VEL
LIN {X 0,Y 340.759,Z 198.852,A -85,B 0,C 180,E1 -14195.638,E2 -14195.638} C_VEL
LIN {X 0,Y 340.74,Z 198.854,A -85,B 0,C 180,E1 -14199.473,E2 -14199.473} C_VEL
LIN {X 0,Y 340.862,Z 198.838,A -85,B 0,C 180,E1 -14201.984,E2 -14201.984} C_VEL
LIN {X 0,Y 340.874,Z 198.839,A -85,B 0,C 180,E1 -14205.704,E2 -14205.704} C_VEL
LIN {X 0,Y 340.852,Z 198.841,A -85,B 0,C 180,E1 -14209.305,E2 -14209.305} C_VEL
LIN {X 0,Y 341.049,Z 198.814,A -85,B 0,C 180,E1 -14212.897,E2 -14212.897} C_VEL
LIN {X 0,Y 341.17,Z 198.799,A -85,B 0,C 180,E1 -14217.638,E2 -14217.638} C_VEL
LIN {X 0,Y 341.278,Z 198.784,A -85,B 0,C 180,E1 -14219.999,E2 -14219.999} C_VEL
LIN {X 0,Y 341.171,Z 198.797,A -85,B 0,C 180,E1 -14222.36,E2 -14222.36} C_VEL
LIN {X 0,Y 341.048,Z 198.817,A -85,B 0,C 180,E1 -14227.101,E2 -14227.101} C_VEL
LIN {X 0,Y 340.85,Z 198.841,A -85,B 0,C 180,E1 -14230.693,E2 -14230.693} C_VEL
LIN {X 0,Y 340.864,Z 198.837,A -85,B 0,C 180,E1 -14234.324,E2 -14234.324} C_VEL
LIN {X 0,Y 340.786,Z 198.849,A -85,B 0,C 180,E1 -14238.439,E2 -14238.439} C_VEL
LIN {X 0,Y 340.717,Z 198.854,A -85,B 0,C 180,E1 -14241.84,E2 -14241.84} C_VEL
LIN {X 0,Y 340.772,Z 198.847,A -85,B 0,C 180,E1 -14245.663,E2 -14245.663} C_VEL
LIN {X 0,Y 340.74,Z 198.856,A -85,B 0,C 180,E1 -14248.318,E2 -14248.318} C_VEL
LIN {X 0,Y 340.702,Z 198.856,A -85,B 0,C 180,E1 -14251.043,E2 -14251.043} C_VEL
LIN {X 0,Y 340.716,Z 198.854,A -85,B 0,C 180,E1 -14255.277,E2 -14255.277} C_VEL
LIN {X 0,Y 340.707,Z 198.858,A -85,B 0,C 180,E1 -14258.385,E2 -14258.385} C_VEL
LIN {X 0,Y 340.695,Z 198.862,A -85,B 0,C 180,E1 -14262.044,E2 -14262.044} C_VEL
LIN {X 0,Y 340.647,Z 198.865,A -85,B 0,C 180,E1 -14266.226,E2 -14266.226} C_VEL
LIN {X 0,Y 340.683,Z 198.863,A -85,B 0,C 180,E1 -14269.752,E2 -14269.752} C_VEL
LIN {X 0,Y 340.7,Z 198.857,A -85,B 0,C 180,E1 -14273.257,E2 -14273.257} C_VEL
LIN {X 0,Y 340.688,Z 198.859,A -85,B 0,C 180,E1 -14276.153,E2 -14276.153} C_VEL
LIN {X 0,Y 340.769,Z 198.848,A -85,B 0,C 180,E1 -14280.332,E2 -14280.332} C_VEL
LIN {X 0,Y 340.798,Z 198.845,A -85,B 0,C 180,E1 -14283.019,E2 -14283.019} C_VEL
LIN {X 0,Y 340.721,Z 198.855,A -85,B 0,C 180,E1 -14286.926,E2 -14286.926} C_VEL
LIN {X 0,Y 340.787,Z 198.846,A -85,B 0,C 180,E1 -14290.733,E2 -14290.733} C_VEL
LIN {X 0,Y 340.78,Z 198.851,A -85,B 0,C 180,E1 -14293.218,E2 -14293.218} C_VEL
LIN {X 0,Y 340.839,Z 198.842,A -85,B 0,C 180,E1 -14296.89,E2 -14296.89} C_VEL
LIN {X 0,Y 340.922,Z 198.829,A -85,B 0,C 180,E1 -14300.507,E2 -14300.507} C_VEL
LIN {X 0,Y 341.067,Z 198.815,A -85,B 0,C 180,E1 -14302.898,E2 -14302.898} C_VEL
LIN {X 0,Y 341.159,Z 198.799,A -85,B 0,C 180,E1 -14307.638,E2 -14307.638} C_VEL
LIN {X 0,Y 341.287,Z 198.783,A -85,B 0,C 180,E1 -14310,E2 -14310} C_VEL
LIN {X 0,Y 341.161,Z 198.801,A -85,B 0,C 180,E1 -14312.361,E2 -14312.361} C_VEL
LIN {X 0,Y 341.069,Z 198.811,A -85,B 0,C 180,E1 -14317.102,E2 -14317.102} C_VEL
LIN {X 0,Y 340.877,Z 198.834,A -85,B 0,C 180,E1 -14319.493,E2 -14319.493} C_VEL
LIN {X 0,Y 340.705,Z 198.856,A -85,B 0,C 180,E1 -14323.115,E2 -14323.115} C_VEL
LIN {X 0,Y 340.385,Z 199.098,A -85,B 0,C 180,E1 -14325.57,E2 -14325.57} C_VEL
LIN {X 0,Y 340.014,Z 203.616,A -85,B 0,C 180,E1 -14329.312,E2 -14329.312} C_VEL
LIN {X 0,Y 339.87,Z 206.759,A -85,B 0,C 180,E1 -14331.852,E2 -14331.852} C_VEL
LIN {X 0,Y 339.743,Z 210.016,A -85,B 0,C 180,E1 -14334.472,E2 -14334.472} C_VEL
LIN {X 0,Y 339.569,Z 213.408,A -85,B 0,C 180,E1 -14337.135,E2 -14337.135} C_VEL
LIN {X 0,Y 339.447,Z 217.471,A -85,B 0,C 180,E1 -14340.18,E2 -14340.18} C_VEL
LIN {X 0,Y 341.27,Z 228.069,A -85,B 0,C 180,E1 -14340.815,E2 -14340.815} C_VEL
LIN {X 0,Y 342.574,Z 237.35,A -85,B 0,C 180,E1 -14341.543,E2 -14341.543} C_VEL
LIN {X 0,Y 342.799,Z 241.026,A -85,B 0,C 180,E1 -14341.865,E2 -14341.865} C_VEL
LIN {X 0,Y 342.169,Z 250.262,A -85,B 0,C 180,E1 -14342.833,E2 -14342.833} C_VEL
LIN {X 0,Y 341.661,Z 257.245,A -85,B 0,C 180,E1 -14343.738,E2 -14343.738} C_VEL
LIN {X 0,Y 341.096,Z 264.284,A -85,B 0,C 180,E1 -14344.846,E2 -14344.846} C_VEL
LIN {X 0,Y 340.554,Z 270.425,A -85,B 0,C 180,E1 -14346.026,E2 -14346.026} C_VEL
LIN {X 0,Y 340.137,Z 276.595,A -85,B 0,C 180,E1 -14347.491,E2 -14347.491} C_VEL
LIN {X 0,Y 339.623,Z 281.85,A -85,B 0,C 180,E1 -14349.135,E2 -14349.135} C_VEL
LIN {X 0,Y 339.311,Z 285.635,A -85,B 0,C 180,E1 -14350.725,E2 -14350.725} C_VEL
LIN {X 0,Y 339.199,Z 287.538,A -85,B 0,C 180,E1 -14351.766,E2 -14351.766} C_VEL
LIN {X 0,Y 339.008,Z 289.626,A -85,B 0,C 180,E1 -14353.484,E2 -14353.484} C_VEL
LIN {X 0,Y 338.969,Z 290.588,A -85,B 0,C 180,E1 -14355.178,E2 -14355.178} C_VEL
LIN {X 0,Y 339.077,Z 290.486,A -85,B 0,C 180,E1 -14356.846,E2 -14356.846} C_VEL
LIN {X 0,Y 339.345,Z 289.34,A -85,B 0,C 180,E1 -14358.493,E2 -14358.493} C_VEL
LIN {X 0,Y 339.666,Z 287.138,A -85,B 0,C 180,E1 -14360.104,E2 -14360.104} C_VEL
LIN {X 0,Y 340.111,Z 283.749,A -85,B 0,C 180,E1 -14361.741,E2 -14361.741} C_VEL
LIN {X 0,Y 340.697,Z 279.494,A -85,B 0,C 180,E1 -14363.259,E2 -14363.259} C_VEL
LIN {X 0,Y 341.24,Z 275.137,A -85,B 0,C 180,E1 -14364.488,E2 -14364.488} C_VEL
LIN {X 0,Y 341.963,Z 269.181,A -85,B 0,C 180,E1 -14365.846,E2 -14365.846} C_VEL
LIN {X 0,Y 342.929,Z 261.121,A -85,B 0,C 180,E1 -14367.295,E2 -14367.295} C_VEL
LIN {X 0,Y 343.409,Z 256.965,A -85,B 0,C 180,E1 -14367.905,E2 -14367.905} C_VEL
LIN {X 0,Y 343.263,Z 252.497,A -85,B 0,C 180,E1 -14368.555,E2 -14368.555} C_VEL
LIN {X 0,Y 342.042,Z 248.042,A -85,B 0,C 180,E1 -14369.187,E2 -14369.187} C_VEL
LIN {X 0,Y 338.203,Z 238.884,A -85,B 0,C 180,E1 -14370.35,E2 -14370.35} C_VEL
LIN {X 0,Y 336.027,Z 232.172,A -85,B 0,C 180,E1 -14371.018,E2 -14371.018} C_VEL
LIN {X 0,Y 333.913,Z 223.295,A -85,B 0,C 180,E1 -14371.735,E2 -14371.735} C_VEL
LIN {X 0,Y 332.768,Z 218.893,A -85,B 0,C 180,E1 -14372.058,E2 -14372.058} C_VEL
LIN {X 0,Y 332.948,Z 215.311,A -85,B 0,C 180,E1 -14375.184,E2 -14375.184} C_VEL
LIN {X 0,Y 333.275,Z 211.07,A -85,B 0,C 180,E1 -14378.994,E2 -14378.994} C_VEL
LIN {X 0,Y 333.562,Z 208.261,A -85,B 0,C 180,E1 -14381.577,E2 -14381.577} C_VEL
LIN {X 0,Y 333.936,Z 204.169,A -85,B 0,C 180,E1 -14385.492,E2 -14385.492} C_VEL
LIN {X 0,Y 333.911,Z 200.666,A -85,B 0,C 180,E1 -14389.082,E2 -14389.082} C_VEL
LIN {X 0,Y 333.825,Z 199.717,A -85,B 0,C 180,E1 -14390.305,E2 -14390.305} C_VEL
LIN {X 0,Y 334.028,Z 199.698,A -85,B 0,C 180,E1 -14392.749,E2 -14392.749} C_VEL
LIN {X 0,Y 333.812,Z 199.725,A -85,B 0,C 180,E1 -14395.17,E2 -14395.17} C_VEL
LIN {X 0,Y 334.106,Z 199.682,A -85,B 0,C 180,E1 -14397.59,E2 -14397.59} C_VEL
LIN {X 0,Y 334.267,Z 199.661,A -85,B 0,C 180,E1 -14400.001,E2 -14400.001} C_VEL
LIN {X 0,Y 334.106,Z 199.682,A -85,B 0,C 180,E1 -14402.412,E2 -14402.412} C_VEL
LIN {X 0,Y 334.011,Z 199.693,A -85,B 0,C 180,E1 -14406.04,E2 -14406.04} C_VEL
LIN {X 0,Y 333.822,Z 199.717,A -85,B 0,C 180,E1 -14409.697,E2 -14409.697} C_VEL
LIN {X 0,Y 333.799,Z 199.719,A -85,B 0,C 180,E1 -14413.392,E2 -14413.392} C_VEL
LIN {X 0,Y 333.749,Z 199.726,A -85,B 0,C 180,E1 -14417.147,E2 -14417.147} C_VEL
LIN {X 0,Y 333.744,Z 199.727,A -85,B 0,C 180,E1 -14419.691,E2 -14419.691} C_VEL
LIN {X 0,Y 333.694,Z 199.733,A -85,B 0,C 180,E1 -14422.279,E2 -14422.279} C_VEL
LIN {X 0,Y 333.738,Z 199.726,A -85,B 0,C 180,E1 -14426.247,E2 -14426.247} C_VEL
LIN {X 0,Y 333.713,Z 199.73,A -85,B 0,C 180,E1 -14428.973,E2 -14428.973} C_VEL
LIN {X 0,Y 333.645,Z 199.737,A -85,B 0,C 180,E1 -14432.588,E2 -14432.588} C_VEL
LIN {X 0,Y 333.678,Z 199.734,A -85,B 0,C 180,E1 -14436.14,E2 -14436.14} C_VEL
LIN {X 0,Y 333.649,Z 199.74,A -85,B 0,C 180,E1 -14439.193,E2 -14439.193} C_VEL
LIN {X 0,Y 333.635,Z 199.743,A -85,B 0,C 180,E1 -14442.5,E2 -14442.5} C_VEL
LIN {X 0,Y 333.599,Z 199.749,A -85,B 0,C 180,E1 -14445.956,E2 -14445.956} C_VEL
LIN {X 0,Y 333.644,Z 199.763,A -85,B 0,C 180,E1 -14447.619,E2 -14447.619} C_VEL
LIN {X 0,Y 334.489,Z 204.034,A -85,B 0,C 180,E1 -14451.025,E2 -14451.025} C_VEL
LIN {X 0,Y 335.45,Z 209.282,A -85,B 0,C 180,E1 -14454.795,E2 -14454.795} C_VEL
LIN {X 0,Y 336.135,Z 213.838,A -85,B 0,C 180,E1 -14457.781,E2 -14457.781} C_VEL
LIN {X 0,Y 335.702,Z 217.346,A -85,B 0,C 180,E1 -14459.838,E2 -14459.838} C_VEL
LIN {X 0,Y 334.728,Z 223.244,A -85,B 0,C 180,E1 -14463.166,E2 -14463.166} C_VEL
LIN {X 0,Y 333.942,Z 229.282,A -85,B 0,C 180,E1 -14466.43,E2 -14466.43} C_VEL
LIN {X 0,Y 333.184,Z 236.676,A -85,B 0,C 180,E1 -14470.276,E2 -14470.276} C_VEL
LIN {X 0,Y 332.866,Z 240.317,A -85,B 0,C 180,E1 -14472.136,E2 -14472.136} C_VEL
LIN {X 0,Y 335.16,Z 253.073,A -85,B 0,C 180,E1 -14472.929,E2 -14472.929} C_VEL
LIN {X 0,Y 336.106,Z 261.682,A -85,B 0,C 180,E1 -14473.604,E2 -14473.604} C_VEL
LIN {X 0,Y 336.588,Z 270.308,A -85,B 0,C 180,E1 -14474.42,E2 -14474.42} C_VEL
LIN {X 0,Y 336.329,Z 278.458,A -85,B 0,C 180,E1 -14475.328,E2 -14475.328} C_VEL
LIN {X 0,Y 335.362,Z 286.294,A -85,B 0,C 180,E1 -14476.364,E2 -14476.364} C_VEL
LIN {X 0,Y 334.521,Z 293.677,A -85,B 0,C 180,E1 -14477.564,E2 -14477.564} C_VEL
LIN {X 0,Y 333.604,Z 301.193,A -85,B 0,C 180,E1 -14479.071,E2 -14479.071} C_VEL
LIN {X 0,Y 332.841,Z 308.081,A -85,B 0,C 180,E1 -14480.888,E2 -14480.888} C_VEL
LIN {X 0,Y 332.351,Z 313.325,A -85,B 0,C 180,E1 -14482.711,E2 -14482.711} C_VEL
LIN {X 0,Y 332.093,Z 316.297,A -85,B 0,C 180,E1 -14484.075,E2 -14484.075} C_VEL
LIN {X 0,Y 332.039,Z 318.133,A -85,B 0,C 180,E1 -14485.143,E2 -14485.143} C_VEL
LIN {X 0,Y 332.039,Z 319.736,A -85,B 0,C 180,E1 -14486.36,E2 -14486.36} C_VEL
LIN {X 0,Y 331.987,Z 320.76,A -85,B 0,C 180,E1 -14487.574,E2 -14487.574} C_VEL
LIN {X 0,Y 332.061,Z 321.22,A -85,B 0,C 180,E1 -14488.787,E2 -14488.787} C_VEL
LIN {X 0,Y 332.134,Z 321.198,A -85,B 0,C 180,E1 -14490,E2 -14490} C_VEL
LIN {X 0,Y 332.1,Z 320.689,A -85,B 0,C 180,E1 -14491.213,E2 -14491.213} C_VEL
LIN {X 0,Y 332.009,Z 319.678,A -85,B 0,C 180,E1 -14492.427,E2 -14492.427} C_VEL
LIN {X 0,Y 332.13,Z 317.024,A -85,B 0,C 180,E1 -14494.248,E2 -14494.248} C_VEL
LIN {X 0,Y 332.142,Z 313.066,A -85,B 0,C 180,E1 -14496.073,E2 -14496.073} C_VEL
LIN {X 0,Y 332.32,Z 309.612,A -85,B 0,C 180,E1 -14497.29,E2 -14497.29} C_VEL
LIN {X 0,Y 332.631,Z 304.235,A -85,B 0,C 180,E1 -14498.812,E2 -14498.812} C_VEL
LIN {X 0,Y 333.149,Z 297.507,A -85,B 0,C 180,E1 -14500.33,E2 -14500.33} C_VEL
LIN {X 0,Y 333.77,Z 288.815,A -85,B 0,C 180,E1 -14501.847,E2 -14501.847} C_VEL
LIN {X 0,Y 334.47,Z 281.242,A -85,B 0,C 180,E1 -14502.901,E2 -14502.901} C_VEL
LIN {X 0,Y 335.044,Z 273.297,A -85,B 0,C 180,E1 -14503.805,E2 -14503.805} C_VEL
LIN {X 0,Y 334.702,Z 264.955,A -85,B 0,C 180,E1 -14504.595,E2 -14504.595} C_VEL
LIN {X 0,Y 334.025,Z 256.42,A -85,B 0,C 180,E1 -14505.248,E2 -14505.248} C_VEL
LIN {X 0,Y 332.959,Z 245.843,A -85,B 0,C 180,E1 -14505.868,E2 -14505.868} C_VEL
LIN {X 0,Y 332.531,Z 241.473,A -85,B 0,C 180,E1 -14506.066,E2 -14506.066} C_VEL
LIN {X 0,Y 332.987,Z 234.12,A -85,B 0,C 180,E1 -14509.737,E2 -14509.737} C_VEL
LIN {X 0,Y 333.667,Z 226.479,A -85,B 0,C 180,E1 -14513.591,E2 -14513.591} C_VEL
LIN {X 0,Y 334.544,Z 218.83,A -85,B 0,C 180,E1 -14517.527,E2 -14517.527} C_VEL
LIN {X 0,Y 335.396,Z 212.664,A -85,B 0,C 180,E1 -14520.78,E2 -14520.78} C_VEL
LIN {X 0,Y 335.435,Z 209.88,A -85,B 0,C 180,E1 -14522.295,E2 -14522.295} C_VEL
LIN {X 0,Y 334.691,Z 205.111,A -85,B 0,C 180,E1 -14525.02,E2 -14525.02} C_VEL
LIN {X 0,Y 333.729,Z 199.729,A -85,B 0,C 180,E1 -14528.311,E2 -14528.311} C_VEL
LIN {X 0,Y 333.637,Z 199.741,A -85,B 0,C 180,E1 -14532.5,E2 -14532.5} C_VEL
LIN {X 0,Y 333.6,Z 199.742,A -85,B 0,C 180,E1 -14535.955,E2 -14535.955} C_VEL
LIN {X 0,Y 333.646,Z 199.734,A -85,B 0,C 180,E1 -14539.316,E2 -14539.316} C_VEL
LIN {X 0,Y 333.667,Z 199.732,A -85,B 0,C 180,E1 -14543.168,E2 -14543.168} C_VEL
LIN {X 0,Y 333.678,Z 199.73,A -85,B 0,C 180,E1 -14545.341,E2 -14545.341} C_VEL
LIN {X 0,Y 333.695,Z 199.731,A -85,B 0,C 180,E1 -14549.637,E2 -14549.637} C_VEL
LIN {X 0,Y 333.744,Z 199.724,A -85,B 0,C 180,E1 -14552.4,E2 -14552.4} C_VEL
LIN {X 0,Y 333.73,Z 199.724,A -85,B 0,C 180,E1 -14555.09,E2 -14555.09} C_VEL
LIN {X 0,Y 333.678,Z 199.731,A -85,B 0,C 180,E1 -14559.018,E2 -14559.018} C_VEL
LIN {X 0,Y 333.799,Z 199.72,A -85,B 0,C 180,E1 -14561.589,E2 -14561.589} C_VEL
LIN {X 0,Y 333.813,Z 199.719,A -85,B 0,C 180,E1 -14565.576,E2 -14565.576} C_VEL
LIN {X 0,Y 333.822,Z 199.715,A -85,B 0,C 180,E1 -14569.077,E2 -14569.077} C_VEL
LIN {X 0,Y 333.996,Z 199.692,A -85,B 0,C 180,E1 -14572.746,E2 -14572.746} C_VEL
LIN {X 0,Y 333.809,Z 199.718,A -85,B 0,C 180,E1 -14575.168,E2 -14575.168} C_VEL
LIN {X 0,Y 334.108,Z 199.679,A -85,B 0,C 180,E1 -14577.588,E2 -14577.588} C_VEL
LIN {X 0,Y 334.229,Z 199.662,A -85,B 0,C 180,E1 -14579.999,E2 -14579.999} C_VEL
LIN {X 0,Y 334.108,Z 199.677,A -85,B 0,C 180,E1 -14582.41,E2 -14582.41} C_VEL
LIN {X 0,Y 333.984,Z 199.691,A -85,B 0,C 180,E1 -14586.636,E2 -14586.636} C_VEL
LIN {X 0,Y 333.822,Z 199.713,A -85,B 0,C 180,E1 -14589.695,E2 -14589.695} C_VEL
LIN {X 0,Y 333.798,Z 199.716,A -85,B 0,C 180,E1 -14593.39,E2 -14593.39} C_VEL
LIN {X 0,Y 333.72,Z 199.727,A -85,B 0,C 180,E1 -14597.146,E2 -14597.146} C_VEL
LIN {X 0,Y 333.672,Z 199.731,A -85,B 0,C 180,E1 -14599.693,E2 -14599.693} C_VEL
LIN {X 0,Y 333.669,Z 199.731,A -85,B 0,C 180,E1 -14603.589,E2 -14603.589} C_VEL
LIN {X 0,Y 333.735,Z 199.727,A -85,B 0,C 180,E1 -14606.245,E2 -14606.245} C_VEL
LIN {X 0,Y 333.71,Z 199.727,A -85,B 0,C 180,E1 -14608.971,E2 -14608.971} C_VEL
LIN {X 0,Y 333.644,Z 199.738,A -85,B 0,C 180,E1 -14612.586,E2 -14612.586} C_VEL
LIN {X 0,Y 333.674,Z 199.736,A -85,B 0,C 180,E1 -14616.138,E2 -14616.138} C_VEL
LIN {X 0,Y 333.644,Z 199.734,A -85,B 0,C 180,E1 -14619.191,E2 -14619.191} C_VEL
LIN {X 0,Y 333.628,Z 199.738,A -85,B 0,C 180,E1 -14622.499,E2 -14622.499} C_VEL
LIN {X 0,Y 333.592,Z 199.747,A -85,B 0,C 180,E1 -14625.954,E2 -14625.954} C_VEL
LIN {X 0,Y 333.642,Z 199.736,A -85,B 0,C 180,E1 -14629.314,E2 -14629.314} C_VEL
LIN {X 0,Y 333.66,Z 199.734,A -85,B 0,C 180,E1 -14633.167,E2 -14633.167} C_VEL
LIN {X 0,Y 333.632,Z 199.736,A -85,B 0,C 180,E1 -14636.791,E2 -14636.791} C_VEL
LIN {X 0,Y 333.696,Z 199.732,A -85,B 0,C 180,E1 -14639.709,E2 -14639.709} C_VEL
LIN {X 0,Y 333.738,Z 199.723,A -85,B 0,C 180,E1 -14642.4,E2 -14642.4} C_VEL
LIN {X 0,Y 333.72,Z 199.728,A -85,B 0,C 180,E1 -14645.09,E2 -14645.09} C_VEL
LIN {X 0,Y 333.675,Z 199.734,A -85,B 0,C 180,E1 -14649.019,E2 -14649.019} C_VEL
LIN {X 0,Y 333.787,Z 199.719,A -85,B 0,C 180,E1 -14651.589,E2 -14651.589} C_VEL
LIN {X 0,Y 333.8,Z 199.717,A -85,B 0,C 180,E1 -14655.576,E2 -14655.576} C_VEL
LIN {X 0,Y 333.83,Z 199.717,A -85,B 0,C 180,E1 -14659.078,E2 -14659.078} C_VEL
LIN {X 0,Y 334.017,Z 199.692,A -85,B 0,C 180,E1 -14662.747,E2 -14662.747} C_VEL
LIN {X 0,Y 333.802,Z 199.718,A -85,B 0,C 180,E1 -14665.169,E2 -14665.169} C_VEL
LIN {X 0,Y 334.096,Z 199.678,A -85,B 0,C 180,E1 -14667.589,E2 -14667.589} C_VEL
LIN {X 0,Y 334.238,Z 199.661,A -85,B 0,C 180,E1 -14670,E2 -14670} C_VEL
LIN {X 0,Y 334.099,Z 199.681,A -85,B 0,C 180,E1 -14672.411,E2 -14672.411} C_VEL
LIN {X 0,Y 334.019,Z 199.688,A -85,B 0,C 180,E1 -14677.252,E2 -14677.252} C_VEL
LIN {X 0,Y 333.813,Z 199.714,A -85,B 0,C 180,E1 -14679.696,E2 -14679.696} C_VEL
LIN {X 0,Y 333.631,Z 199.736,A -85,B 0,C 180,E1 -14683.398,E2 -14683.398} C_VEL
LIN {X 0,Y 333.331,Z 199.975,A -85,B 0,C 180,E1 -14685.594,E2 -14685.594} C_VEL
LIN {X 0,Y 332.935,Z 204.923,A -85,B 0,C 180,E1 -14689.74,E2 -14689.74} C_VEL
LIN {X 0,Y 332.751,Z 208.096,A -85,B 0,C 180,E1 -14692.344,E2 -14692.344} C_VEL
LIN {X 0,Y 332.641,Z 211.387,A -85,B 0,C 180,E1 -14694.996,E2 -14694.996} C_VEL
LIN {X 0,Y 332.427,Z 214.777,A -85,B 0,C 180,E1 -14697.717,E2 -14697.717} C_VEL
LIN {X 0,Y 332.369,Z 217.53,A -85,B 0,C 180,E1 -14699.897,E2 -14699.897} C_VEL
LIN {X 0,Y 334.366,Z 229.356,A -85,B 0,C 180,E1 -14700.644,E2 -14700.644} C_VEL
LIN {X 0,Y 335.634,Z 238.46,A -85,B 0,C 180,E1 -14701.39,E2 -14701.39} C_VEL
LIN {X 0,Y 335.757,Z 242.121,A -85,B 0,C 180,E1 -14701.729,E2 -14701.729} C_VEL
LIN {X 0,Y 335.171,Z 250.885,A -85,B 0,C 180,E1 -14702.679,E2 -14702.679} C_VEL
LIN {X 0,Y 334.623,Z 258.062,A -85,B 0,C 180,E1 -14703.638,E2 -14703.638} C_VEL
LIN {X 0,Y 333.97,Z 265.463,A -85,B 0,C 180,E1 -14704.847,E2 -14704.847} C_VEL
LIN {X 0,Y 333.388,Z 273.207,A -85,B 0,C 180,E1 -14706.453,E2 -14706.453} C_VEL
LIN {X 0,Y 332.787,Z 279.475,A -85,B 0,C 180,E1 -14708.17,E2 -14708.17} C_VEL
LIN {X 0,Y 332.375,Z 284.239,A -85,B 0,C 180,E1 -14709.88,E2 -14709.88} C_VEL
LIN {X 0,Y 332.178,Z 286.521,A -85,B 0,C 180,E1 -14710.986,E2 -14710.986} C_VEL
LIN {X 0,Y 331.994,Z 289.087,A -85,B 0,C 180,E1 -14712.641,E2 -14712.641} C_VEL
LIN {X 0,Y 331.896,Z 290.61,A -85,B 0,C 180,E1 -14714.329,E2 -14714.329} C_VEL
LIN {X 0,Y 331.926,Z 291.023,A -85,B 0,C 180,E1 -14716.046,E2 -14716.046} C_VEL
LIN {X 0,Y 332.106,Z 290.342,A -85,B 0,C 180,E1 -14717.788,E2 -14717.788} C_VEL
LIN {X 0,Y 332.464,Z 288.536,A -85,B 0,C 180,E1 -14719.553,E2 -14719.553} C_VEL
LIN {X 0,Y 332.914,Z 285.488,A -85,B 0,C 180,E1 -14721.36,E2 -14721.36} C_VEL
LIN {X 0,Y 333.598,Z 280.857,A -85,B 0,C 180,E1 -14723.183,E2 -14723.183} C_VEL
LIN {X 0,Y 334.185,Z 276.434,A -85,B 0,C 180,E1 -14724.516,E2 -14724.516} C_VEL
LIN {X 0,Y 334.918,Z 270.912,A -85,B 0,C 180,E1 -14725.851,E2 -14725.851} C_VEL
LIN {X 0,Y 335.801,Z 263.905,A -85,B 0,C 180,E1 -14727.213,E2 -14727.213} C_VEL
LIN {X 0,Y 336.944,Z 254.984,A -85,B 0,C 180,E1 -14728.572,E2 -14728.572} C_VEL
LIN {X 0,Y 337.606,Z 247.204,A -85,B 0,C 180,E1 -14729.51,E2 -14729.51} C_VEL
LIN {X 0,Y 337.896,Z 243.596,A -85,B 0,C 180,E1 -14729.884,E2 -14729.884} C_VEL
LIN {X 0,Y 336.261,Z 233.221,A -85,B 0,C 180,E1 -14730.928,E2 -14730.928} C_VEL
LIN {X 0,Y 336.027,Z 232.172,A -85,B 0,C 180,E1 -14731.018,E2 -14731.018} C_VEL
LIN {X 0,Y 335.001,Z 229.003,A -85,B 0,C 180,E1 -14731.342,E2 -14731.342} C_VEL
LIN {X 0,Y 332.758,Z 224.98,A -85,B 0,C 180,E1 -14731.941,E2 -14731.941} C_VEL
LIN {X 0,Y 329.381,Z 220.839,A -85,B 0,C 180,E1 -14732.912,E2 -14732.912} C_VEL
LIN {X 0,Y 326.673,Z 217.893,A -85,B 0,C 180,E1 -14734.068,E2 -14734.068} C_VEL
LIN {X 0,Y 325.896,Z 216.433,A -85,B 0,C 180,E1 -14735.036,E2 -14735.036} C_VEL
LIN {X 0,Y 326.225,Z 212.602,A -85,B 0,C 180,E1 -14738.518,E2 -14738.518} C_VEL
LIN {X 0,Y 326.595,Z 208.433,A -85,B 0,C 180,E1 -14742.468,E2 -14742.468} C_VEL
LIN {X 0,Y 326.902,Z 205.523,A -85,B 0,C 180,E1 -14745.34,E2 -14745.34} C_VEL
LIN {X 0,Y 326.935,Z 202.166,A -85,B 0,C 180,E1 -14748.846,E2 -14748.846} C_VEL
LIN {X 0,Y 326.841,Z 201.028,A -85,B 0,C 180,E1 -14750.096,E2 -14750.096} C_VEL
LIN {X 0,Y 326.923,Z 200.58,A -85,B 0,C 180,E1 -14751.448,E2 -14751.448} C_VEL
LIN {X 0,Y 326.997,Z 200.575,A -85,B 0,C 180,E1 -14753.832,E2 -14753.832} C_VEL
LIN {X 0,Y 327.047,Z 200.562,A -85,B 0,C 180,E1 -14757.538,E2 -14757.538} C_VEL
LIN {X 0,Y 327.218,Z 200.54,A -85,B 0,C 180,E1 -14760.001,E2 -14760.001} C_VEL
LIN {X 0,Y 327.047,Z 200.561,A -85,B 0,C 180,E1 -14762.464,E2 -14762.464} C_VEL
LIN {X 0,Y 326.985,Z 200.568,A -85,B 0,C 180,E1 -14766.17,E2 -14766.17} C_VEL
LIN {X 0,Y 326.785,Z 200.593,A -85,B 0,C 180,E1 -14769.908,E2 -14769.908} C_VEL
LIN {X 0,Y 326.761,Z 200.596,A -85,B 0,C 180,E1 -14773.686,E2 -14773.686} C_VEL
LIN {X 0,Y 326.702,Z 200.603,A -85,B 0,C 180,E1 -14777.529,E2 -14777.529} C_VEL
LIN {X 0,Y 326.67,Z 200.607,A -85,B 0,C 180,E1 -14780.135,E2 -14780.135} C_VEL
LIN {X 0,Y 326.654,Z 200.61,A -85,B 0,C 180,E1 -14784.13,E2 -14784.13} C_VEL
LIN {X 0,Y 326.686,Z 200.606,A -85,B 0,C 180,E1 -14786.858,E2 -14786.858} C_VEL
LIN {X 0,Y 326.641,Z 200.61,A -85,B 0,C 180,E1 -14790.612,E2 -14790.612} C_VEL
LIN {X 0,Y 326.609,Z 200.613,A -85,B 0,C 180,E1 -14794.02,E2 -14794.02} C_VEL
LIN {X 0,Y 326.63,Z 200.612,A -85,B 0,C 180,E1 -14797.239,E2 -14797.239} C_VEL
LIN {X 0,Y 326.58,Z 200.622,A -85,B 0,C 180,E1 -14801.132,E2 -14801.132} C_VEL
LIN {X 0,Y 326.53,Z 200.629,A -85,B 0,C 180,E1 -14804.743,E2 -14804.743} C_VEL
LIN {X 0,Y 326.578,Z 200.747,A -85,B 0,C 180,E1 -14807.029,E2 -14807.029} C_VEL
LIN {X 0,Y 327.471,Z 205.013,A -85,B 0,C 180,E1 -14810.59,E2 -14810.59} C_VEL
LIN {X 0,Y 328.415,Z 210.141,A -85,B 0,C 180,E1 -14814.41,E2 -14814.41} C_VEL
LIN {X 0,Y 329.169,Z 215.077,A -85,B 0,C 180,E1 -14817.74,E2 -14817.74} C_VEL
LIN {X 0,Y 328.495,Z 219.723,A -85,B 0,C 180,E1 -14820.523,E2 -14820.523} C_VEL
LIN {X 0,Y 327.345,Z 226.837,A -85,B 0,C 180,E1 -14824.571,E2 -14824.571} C_VEL
LIN {X 0,Y 326.455,Z 234.116,A -85,B 0,C 180,E1 -14828.532,E2 -14828.532} C_VEL
LIN {X 0,Y 325.868,Z 239.98,A -85,B 0,C 180,E1 -14831.615,E2 -14831.615} C_VEL
LIN {X 0,Y 328.214,Z 252.592,A -85,B 0,C 180,E1 -14832.448,E2 -14832.448} C_VEL
LIN {X 0,Y 329.209,Z 261.082,A -85,B 0,C 180,E1 -14833.138,E2 -14833.138} C_VEL
LIN {X 0,Y 329.723,Z 270.13,A -85,B 0,C 180,E1 -14834.023,E2 -14834.023} C_VEL
LIN {X 0,Y 329.568,Z 277.618,A -85,B 0,C 180,E1 -14834.876,E2 -14834.876} C_VEL
LIN {X 0,Y 328.596,Z 285.449,A -85,B 0,C 180,E1 -14835.919,E2 -14835.919} C_VEL
LIN {X 0,Y 327.767,Z 292.064,A -85,B 0,C 180,E1 -14836.989,E2 -14836.989} C_VEL
LIN {X 0,Y 327.002,Z 298.365,A -85,B 0,C 180,E1 -14838.219,E2 -14838.219} C_VEL
LIN {X 0,Y 326.311,Z 303.611,A -85,B 0,C 180,E1 -14839.452,E2 -14839.452} C_VEL
LIN {X 0,Y 325.827,Z 307.992,A -85,B 0,C 180,E1 -14840.69,E2 -14840.69} C_VEL
LIN {X 0,Y 325.294,Z 313.188,A -85,B 0,C 180,E1 -14842.552,E2 -14842.552} C_VEL
LIN {X 0,Y 325,Z 316.45,A -85,B 0,C 180,E1 -14844.122,E2 -14844.122} C_VEL
LIN {X 0,Y 324.964,Z 319.465,A -85,B 0,C 180,E1 -14846.28,E2 -14846.28} C_VEL
LIN {X 0,Y 324.904,Z 320.479,A -85,B 0,C 180,E1 -14847.521,E2 -14847.521} C_VEL
LIN {X 0,Y 324.963,Z 320.908,A -85,B 0,C 180,E1 -14848.761,E2 -14848.761} C_VEL
LIN {X 0,Y 325.042,Z 320.85,A -85,B 0,C 180,E1 -14850,E2 -14850} C_VEL
LIN {X 0,Y 325.004,Z 320.303,A -85,B 0,C 180,E1 -14851.239,E2 -14851.239} C_VEL
LIN {X 0,Y 324.925,Z 319.258,A -85,B 0,C 180,E1 -14852.48,E2 -14852.48} C_VEL
LIN {X 0,Y 325.035,Z 316.558,A -85,B 0,C 180,E1 -14854.34,E2 -14854.34} C_VEL
LIN {X 0,Y 325.028,Z 313.238,A -85,B 0,C 180,E1 -14855.927,E2 -14855.927} C_VEL
LIN {X 0,Y 325.271,Z 309.053,A -85,B 0,C 180,E1 -14857.449,E2 -14857.449} C_VEL
LIN {X 0,Y 325.602,Z 303.621,A -85,B 0,C 180,E1 -14859.003,E2 -14859.003} C_VEL
LIN {X 0,Y 326.125,Z 296.818,A -85,B 0,C 180,E1 -14860.555,E2 -14860.555} C_VEL
LIN {X 0,Y 326.812,Z 287.98,A -85,B 0,C 180,E1 -14862.103,E2 -14862.103} C_VEL
LIN {X 0,Y 327.552,Z 280.304,A -85,B 0,C 180,E1 -14863.178,E2 -14863.178} C_VEL
LIN {X 0,Y 328.051,Z 272.235,A -85,B 0,C 180,E1 -14864.102,E2 -14864.102} C_VEL
LIN {X 0,Y 327.473,Z 262.344,A -85,B 0,C 180,E1 -14865.035,E2 -14865.035} C_VEL
LIN {X 0,Y 326.396,Z 250.339,A -85,B 0,C 180,E1 -14865.874,E2 -14865.874} C_VEL
LIN {X 0,Y 325.466,Z 241.194,A -85,B 0,C 180,E1 -14866.344,E2 -14866.344} C_VEL
LIN {X 0,Y 325.981,Z 233.705,A -85,B 0,C 180,E1 -14870.179,E2 -14870.179} C_VEL
LIN {X 0,Y 326.694,Z 226.106,A -85,B 0,C 180,E1 -14874.126,E2 -14874.126} C_VEL
LIN {X 0,Y 327.651,Z 218.478,A -85,B 0,C 180,E1 -14878.158,E2 -14878.158} C_VEL
LIN {X 0,Y 328.52,Z 212.003,A -85,B 0,C 180,E1 -14881.663,E2 -14881.663} C_VEL
LIN {X 0,Y 327.827,Z 206.925,A -85,B 0,C 180,E1 -14884.61,E2 -14884.61} C_VEL
LIN {X 0,Y 326.664,Z 200.609,A -85,B 0,C 180,E1 -14888.518,E2 -14888.518} C_VEL
LIN {X 0,Y 326.58,Z 200.615,A -85,B 0,C 180,E1 -14891.846,E2 -14891.846} C_VEL
LIN {X 0,Y 326.531,Z 200.621,A -85,B 0,C 180,E1 -14895.257,E2 -14895.257} C_VEL
LIN {X 0,Y 326.578,Z 200.616,A -85,B 0,C 180,E1 -14898.869,E2 -14898.869} C_VEL
LIN {X 0,Y 326.627,Z 200.609,A -85,B 0,C 180,E1 -14902.762,E2 -14902.762} C_VEL
LIN {X 0,Y 326.611,Z 200.615,A -85,B 0,C 180,E1 -14905.98,E2 -14905.98} C_VEL
LIN {X 0,Y 326.652,Z 200.608,A -85,B 0,C 180,E1 -14910.339,E2 -14910.339} C_VEL
LIN {X 0,Y 326.694,Z 200.601,A -85,B 0,C 180,E1 -14914.516,E2 -14914.516} C_VEL
LIN {X 0,Y 326.624,Z 200.609,A -85,B 0,C 180,E1 -14918.543,E2 -14918.543} C_VEL
LIN {X 0,Y 326.749,Z 200.595,A -85,B 0,C 180,E1 -14921.177,E2 -14921.177} C_VEL
LIN {X 0,Y 326.767,Z 200.595,A -85,B 0,C 180,E1 -14925.432,E2 -14925.432} C_VEL
LIN {X 0,Y 326.763,Z 200.592,A -85,B 0,C 180,E1 -14928.838,E2 -14928.838} C_VEL
LIN {X 0,Y 326.946,Z 200.569,A -85,B 0,C 180,E1 -14932.589,E2 -14932.589} C_VEL
LIN {X 0,Y 326.986,Z 200.565,A -85,B 0,C 180,E1 -14933.83,E2 -14933.83} C_VEL
LIN {X 0,Y 327.048,Z 200.559,A -85,B 0,C 180,E1 -14937.536,E2 -14937.536} C_VEL
LIN {X 0,Y 327.181,Z 200.54,A -85,B 0,C 180,E1 -14939.999,E2 -14939.999} C_VEL
LIN {X 0,Y 327.049,Z 200.557,A -85,B 0,C 180,E1 -14942.462,E2 -14942.462} C_VEL
LIN {X 0,Y 326.952,Z 200.567,A -85,B 0,C 180,E1 -14946.626,E2 -14946.626} C_VEL
LIN {X 0,Y 326.785,Z 200.589,A -85,B 0,C 180,E1 -14949.906,E2 -14949.906} C_VEL
LIN {X 0,Y 326.761,Z 200.592,A -85,B 0,C 180,E1 -14953.684,E2 -14953.684} C_VEL
LIN {X 0,Y 326.664,Z 200.604,A -85,B 0,C 180,E1 -14957.529,E2 -14957.529} C_VEL
LIN {X 0,Y 326.618,Z 200.61,A -85,B 0,C 180,E1 -14961.455,E2 -14961.455} C_VEL
LIN {X 0,Y 326.689,Z 200.601,A -85,B 0,C 180,E1 -14965.482,E2 -14965.482} C_VEL
LIN {X 0,Y 326.659,Z 200.605,A -85,B 0,C 180,E1 -14969.658,E2 -14969.658} C_VEL
LIN {X 0,Y 326.605,Z 200.614,A -85,B 0,C 180,E1 -14974.018,E2 -14974.018} C_VEL
LIN {X 0,Y 326.625,Z 200.609,A -85,B 0,C 180,E1 -14977.237,E2 -14977.237} C_VEL
LIN {X 0,Y 326.574,Z 200.615,A -85,B 0,C 180,E1 -14981.13,E2 -14981.13} C_VEL
LIN {X 0,Y 326.523,Z 200.622,A -85,B 0,C 180,E1 -14984.741,E2 -14984.741} C_VEL
LIN {X 0,Y 326.571,Z 200.618,A -85,B 0,C 180,E1 -14988.153,E2 -14988.153} C_VEL
LIN {X 0,Y 326.618,Z 200.612,A -85,B 0,C 180,E1 -14991.39,E2 -14991.39} C_VEL
LIN {X 0,Y 326.613,Z 200.61,A -85,B 0,C 180,E1 -14994.85,E2 -14994.85} C_VEL
LIN {X 0,Y 326.604,Z 200.615,A -85,B 0,C 180,E1 -14997.455,E2 -14997.455} C_VEL
LIN {X 0,Y 326.654,Z 200.605,A -85,B 0,C 180,E1 -15000.34,E2 -15000.34} C_VEL
LIN {X 0,Y 326.683,Z 200.601,A -85,B 0,C 180,E1 -15004.515,E2 -15004.515} C_VEL
LIN {X 0,Y 326.639,Z 200.607,A -85,B 0,C 180,E1 -15008.545,E2 -15008.545} C_VEL
LIN {X 0,Y 326.737,Z 200.6,A -85,B 0,C 180,E1 -15011.177,E2 -15011.177} C_VEL
LIN {X 0,Y 326.755,Z 200.595,A -85,B 0,C 180,E1 -15015.432,E2 -15015.432} C_VEL
LIN {X 0,Y 326.766,Z 200.595,A -85,B 0,C 180,E1 -15018.839,E2 -15018.839} C_VEL
LIN {X 0,Y 326.971,Z 200.568,A -85,B 0,C 180,E1 -15022.59,E2 -15022.59} C_VEL
LIN {X 0,Y 326.769,Z 200.595,A -85,B 0,C 180,E1 -15025.064,E2 -15025.064} C_VEL
LIN {X 0,Y 327.037,Z 200.558,A -85,B 0,C 180,E1 -15027.536,E2 -15027.536} C_VEL
LIN {X 0,Y 327.19,Z 200.539,A -85,B 0,C 180,E1 -15030,E2 -15030} C_VEL
LIN {X 0,Y 327.039,Z 200.561,A -85,B 0,C 180,E1 -15032.463,E2 -15032.463} C_VEL
LIN {X 0,Y 326.988,Z 200.565,A -85,B 0,C 180,E1 -15036.169,E2 -15036.169} C_VEL
LIN {X 0,Y 326.951,Z 200.572,A -85,B 0,C 180,E1 -15038.654,E2 -15038.654} C_VEL
LIN {X 0,Y 326.64,Z 200.612,A -85,B 0,C 180,E1 -15042.425,E2 -15042.425} C_VEL
LIN {X 0,Y 326.327,Z 200.659,A -85,B 0,C 180,E1 -15045.457,E2 -15045.457} C_VEL
LIN {X 0,Y 325.841,Z 206.23,A -85,B 0,C 180,E1 -15050.188,E2 -15050.188} C_VEL
LIN {X 0,Y 325.613,Z 211.076,A -85,B 0,C 180,E1 -15054.211,E2 -15054.211} C_VEL
LIN {X 0,Y 325.356,Z 215.359,A -85,B 0,C 180,E1 -15057.673,E2 -15057.673} C_VEL
LIN {X 0,Y 325.305,Z 217.936,A -85,B 0,C 180,E1 -15059.661,E2 -15059.661} C_VEL
LIN {X 0,Y 326.981,Z 227.797,A -85,B 0,C 180,E1 -15060.267,E2 -15060.267} C_VEL
LIN {X 0,Y 328.224,Z 236.073,A -85,B 0,C 180,E1 -15060.923,E2 -15060.923} C_VEL
LIN {X 0,Y 328.777,Z 242.359,A -85,B 0,C 180,E1 -15061.51,E2 -15061.51} C_VEL
LIN {X 0,Y 328.23,Z 250.209,A -85,B 0,C 180,E1 -15062.364,E2 -15062.364} C_VEL
LIN {X 0,Y 327.716,Z 256.888,A -85,B 0,C 180,E1 -15063.244,E2 -15063.244} C_VEL
LIN {X 0,Y 327.13,Z 263.694,A -85,B 0,C 180,E1 -15064.329,E2 -15064.329} C_VEL
LIN {X 0,Y 326.566,Z 269.874,A -85,B 0,C 180,E1 -15065.525,E2 -15065.525} C_VEL
LIN {X 0,Y 326.197,Z 274.923,A -85,B 0,C 180,E1 -15066.708,E2 -15066.708} C_VEL
LIN {X 0,Y 325.767,Z 279.291,A -85,B 0,C 180,E1 -15067.941,E2 -15067.941} C_VEL
LIN {X 0,Y 325.482,Z 282.393,A -85,B 0,C 180,E1 -15068.985,E2 -15068.985} C_VEL
LIN {X 0,Y 325.101,Z 286.57,A -85,B 0,C 180,E1 -15070.835,E2 -15070.835} C_VEL
LIN {X 0,Y 324.897,Z 289.396,A -85,B 0,C 180,E1 -15072.655,E2 -15072.655} C_VEL
LIN {X 0,Y 324.798,Z 290.964,A -85,B 0,C 180,E1 -15074.436,E2 -15074.436} C_VEL
LIN {X 0,Y 324.841,Z 291.35,A -85,B 0,C 180,E1 -15076.187,E2 -15076.187} C_VEL
LIN {X 0,Y 325.036,Z 290.691,A -85,B 0,C 180,E1 -15077.913,E2 -15077.913} C_VEL
LIN {X 0,Y 325.39,Z 289.025,A -85,B 0,C 180,E1 -15079.614,E2 -15079.614} C_VEL
LIN {X 0,Y 325.818,Z 286.371,A -85,B 0,C 180,E1 -15081.28,E2 -15081.28} C_VEL
LIN {X 0,Y 326.438,Z 282.646,A -85,B 0,C 180,E1 -15082.93,E2 -15082.93} C_VEL
LIN {X 0,Y 327.206,Z 277.13,A -85,B 0,C 180,E1 -15084.706,E2 -15084.706} C_VEL
LIN {X 0,Y 328.051,Z 271.302,A -85,B 0,C 180,E1 -15086.152,E2 -15086.152} C_VEL
LIN {X 0,Y 328.975,Z 264.349,A -85,B 0,C 180,E1 -15087.539,E2 -15087.539} C_VEL
LIN {X 0,Y 330.162,Z 255.631,A -85,B 0,C 180,E1 -15088.907,E2 -15088.907} C_VEL
LIN {X 0,Y 330.877,Z 247.779,A -85,B 0,C 180,E1 -15089.882,E2 -15089.882} C_VEL
LIN {X 0,Y 331.066,Z 244.202,A -85,B 0,C 180,E1 -15090.27,E2 -15090.27} C_VEL
LIN {X 0,Y 329.467,Z 234.257,A -85,B 0,C 180,E1 -15091.319,E2 -15091.319} C_VEL
LIN {X 0,Y 327.004,Z 223.859,A -85,B 0,C 180,E1 -15092.198,E2 -15092.198} C_VEL
LIN {X 0,Y 325.752,Z 219.194,A -85,B 0,C 180,E1 -15092.56,E2 -15092.56} C_VEL
LIN {X 0,Y 325.896,Z 216.433,A -85,B 0,C 180,E1 -15095.036,E2 -15095.036} C_VEL
LIN {X 0,Y 325.276,Z 215.401,A -85,B 0,C 180,E1 -15096.053,E2 -15096.053} C_VEL
LIN {X 0,Y 322.55,Z 213.989,A -85,B 0,C 180,E1 -15097.721,E2 -15097.721} C_VEL
LIN {X 0,Y 320.284,Z 212.909,A -85,B 0,C 180,E1 -15099.073,E2 -15099.073} C_VEL
LIN {X 0,Y 319.389,Z 211.972,A -85,B 0,C 180,E1 -15100.114,E2 -15100.114} C_VEL
LIN {X 0,Y 319.357,Z 211.62,A -85,B 0,C 180,E1 -15100.464,E2 -15100.464} C_VEL
LIN {X 0,Y 319.675,Z 208.627,A -85,B 0,C 180,E1 -15103.394,E2 -15103.394} C_VEL
LIN {X 0,Y 319.929,Z 206.068,A -85,B 0,C 180,E1 -15106.018,E2 -15106.018} C_VEL
LIN {X 0,Y 319.966,Z 203.674,A -85,B 0,C 180,E1 -15108.6,E2 -15108.6} C_VEL
LIN {X 0,Y 319.88,Z 201.457,A -85,B 0,C 180,E1 -15111.372,E2 -15111.372} C_VEL
LIN {X 0,Y 319.953,Z 201.452,A -85,B 0,C 180,E1 -15113.696,E2 -15113.696} C_VEL
LIN {X 0,Y 319.991,Z 201.441,A -85,B 0,C 180,E1 -15117.484,E2 -15117.484} C_VEL
LIN {X 0,Y 320.169,Z 201.418,A -85,B 0,C 180,E1 -15120.001,E2 -15120.001} C_VEL
LIN {X 0,Y 319.991,Z 201.439,A -85,B 0,C 180,E1 -15122.519,E2 -15122.519} C_VEL
LIN {X 0,Y 319.939,Z 201.446,A -85,B 0,C 180,E1 -15126.307,E2 -15126.307} C_VEL
LIN {X 0,Y 319.737,Z 201.471,A -85,B 0,C 180,E1 -15130.129,E2 -15130.129} C_VEL
LIN {X 0,Y 319.734,Z 201.472,A -85,B 0,C 180,E1 -15133.993,E2 -15133.993} C_VEL
LIN {X 0,Y 319.661,Z 201.48,A -85,B 0,C 180,E1 -15137.928,E2 -15137.928} C_VEL
LIN {X 0,Y 319.62,Z 201.485,A -85,B 0,C 180,E1 -15140.599,E2 -15140.599} C_VEL
LIN {X 0,Y 319.572,Z 201.491,A -85,B 0,C 180,E1 -15143.32,E2 -15143.32} C_VEL
LIN {X 0,Y 319.637,Z 201.481,A -85,B 0,C 180,E1 -15146.089,E2 -15146.089} C_VEL
LIN {X 0,Y 319.591,Z 201.489,A -85,B 0,C 180,E1 -15148.934,E2 -15148.934} C_VEL
LIN {X 0,Y 319.534,Z 201.495,A -85,B 0,C 180,E1 -15151.862,E2 -15151.862} C_VEL
LIN {X 0,Y 319.582,Z 201.49,A -85,B 0,C 180,E1 -15155.544,E2 -15155.544} C_VEL
LIN {X 0,Y 319.575,Z 201.493,A -85,B 0,C 180,E1 -15158.009,E2 -15158.009} C_VEL
LIN {X 0,Y 319.528,Z 201.5,A -85,B 0,C 180,E1 -15161.598,E2 -15161.598} C_VEL
LIN {X 0,Y 319.49,Z 201.506,A -85,B 0,C 180,E1 -15165.258,E2 -15165.258} C_VEL
LIN {X 0,Y 319.544,Z 201.669,A -85,B 0,C 180,E1 -15166.361,E2 -15166.361} C_VEL
LIN {X 0,Y 320.528,Z 206.491,A -85,B 0,C 180,E1 -15170.516,E2 -15170.516} C_VEL
LIN {X 0,Y 321.341,Z 211.037,A -85,B 0,C 180,E1 -15174.021,E2 -15174.021} C_VEL
LIN {X 0,Y 322.034,Z 215.194,A -85,B 0,C 180,E1 -15176.935,E2 -15176.935} C_VEL
LIN {X 0,Y 322.058,Z 217.473,A -85,B 0,C 180,E1 -15178.417,E2 -15178.417} C_VEL
LIN {X 0,Y 321.029,Z 223.277,A -85,B 0,C 180,E1 -15181.922,E2 -15181.922} C_VEL
LIN {X 0,Y 319.931,Z 230.43,A -85,B 0,C 180,E1 -15186.022,E2 -15186.022} C_VEL
LIN {X 0,Y 319.082,Z 237.738,A -85,B 0,C 180,E1 -15190.038,E2 -15190.038} C_VEL
LIN {X 0,Y 318.87,Z 239.725,A -85,B 0,C 180,E1 -15191.114,E2 -15191.114} C_VEL
LIN {X 0,Y 321.216,Z 251.777,A -85,B 0,C 180,E1 -15191.914,E2 -15191.914} C_VEL
LIN {X 0,Y 322.412,Z 261.842,A -85,B 0,C 180,E1 -15192.772,E2 -15192.772} C_VEL
LIN {X 0,Y 322.916,Z 271.011,A -85,B 0,C 180,E1 -15193.714,E2 -15193.714} C_VEL
LIN {X 0,Y 322.727,Z 278.055,A -85,B 0,C 180,E1 -15194.556,E2 -15194.556} C_VEL
LIN {X 0,Y 321.74,Z 285.682,A -85,B 0,C 180,E1 -15195.613,E2 -15195.613} C_VEL
LIN {X 0,Y 320.852,Z 292.188,A -85,B 0,C 180,E1 -15196.703,E2 -15196.703} C_VEL
LIN {X 0,Y 320.065,Z 298.398,A -85,B 0,C 180,E1 -15197.96,E2 -15197.96} C_VEL
LIN {X 0,Y 319.334,Z 303.577,A -85,B 0,C 180,E1 -15199.218,E2 -15199.218} C_VEL
LIN {X 0,Y 318.82,Z 307.904,A -85,B 0,C 180,E1 -15200.484,E2 -15200.484} C_VEL
LIN {X 0,Y 318.389,Z 311.5,A -85,B 0,C 180,E1 -15201.751,E2 -15201.751} C_VEL
LIN {X 0,Y 317.971,Z 315.643,A -85,B 0,C 180,E1 -15203.655,E2 -15203.655} C_VEL
LIN {X 0,Y 317.861,Z 317.677,A -85,B 0,C 180,E1 -15204.926,E2 -15204.926} C_VEL
LIN {X 0,Y 317.869,Z 319.196,A -85,B 0,C 180,E1 -15206.197,E2 -15206.197} C_VEL
LIN {X 0,Y 317.823,Z 320.195,A -85,B 0,C 180,E1 -15207.465,E2 -15207.465} C_VEL
LIN {X 0,Y 317.866,Z 320.6,A -85,B 0,C 180,E1 -15208.733,E2 -15208.733} C_VEL
LIN {X 0,Y 317.95,Z 320.496,A -85,B 0,C 180,E1 -15210,E2 -15210} C_VEL
LIN {X 0,Y 317.908,Z 319.905,A -85,B 0,C 180,E1 -15211.267,E2 -15211.267} C_VEL
LIN {X 0,Y 317.844,Z 318.815,A -85,B 0,C 180,E1 -15212.535,E2 -15212.535} C_VEL
LIN {X 0,Y 317.937,Z 317.19,A -85,B 0,C 180,E1 -15213.803,E2 -15213.803} C_VEL
LIN {X 0,Y 317.923,Z 313.178,A -85,B 0,C 180,E1 -15215.858,E2 -15215.858} C_VEL
LIN {X 0,Y 318.209,Z 308.455,A -85,B 0,C 180,E1 -15217.615,E2 -15217.615} C_VEL
LIN {X 0,Y 318.58,Z 302.963,A -85,B 0,C 180,E1 -15219.204,E2 -15219.204} C_VEL
LIN {X 0,Y 319.105,Z 296.052,A -85,B 0,C 180,E1 -15220.79,E2 -15220.79} C_VEL
LIN {X 0,Y 319.758,Z 288.087,A -85,B 0,C 180,E1 -15222.213,E2 -15222.213} C_VEL
LIN {X 0,Y 320.511,Z 280.498,A -85,B 0,C 180,E1 -15223.311,E2 -15223.311} C_VEL
LIN {X 0,Y 321.003,Z 272.855,A -85,B 0,C 180,E1 -15224.222,E2 -15224.222} C_VEL
LIN {X 0,Y 320.516,Z 263.93,A -85,B 0,C 180,E1 -15225.105,E2 -15225.105} C_VEL
LIN {X 0,Y 319.731,Z 254.194,A -85,B 0,C 180,E1 -15225.866,E2 -15225.866} C_VEL
LIN {X 0,Y 318.441,Z 241.51,A -85,B 0,C 180,E1 -15226.57,E2 -15226.57} C_VEL
LIN {X 0,Y 318.399,Z 240.997,A -85,B 0,C 180,E1 -15226.593,E2 -15226.593} C_VEL
LIN {X 0,Y 318.857,Z 234.558,A -85,B 0,C 180,E1 -15229.977,E2 -15229.977} C_VEL
LIN {X 0,Y 319.448,Z 228.239,A -85,B 0,C 180,E1 -15233.329,E2 -15233.329} C_VEL
LIN {X 0,Y 320.408,Z 220.629,A -85,B 0,C 180,E1 -15237.428,E2 -15237.428} C_VEL
LIN {X 0,Y 321.446,Z 213.28,A -85,B 0,C 180,E1 -15241.494,E2 -15241.494} C_VEL
LIN {X 0,Y 321.082,Z 209.477,A -85,B 0,C 180,E1 -15243.719,E2 -15243.719} C_VEL
LIN {X 0,Y 319.859,Z 202.596,A -85,B 0,C 180,E1 -15247.968,E2 -15247.968} C_VEL
LIN {X 0,Y 319.634,Z 201.486,A -85,B 0,C 180,E1 -15248.804,E2 -15248.804} C_VEL
LIN {X 0,Y 319.558,Z 201.49,A -85,B 0,C 180,E1 -15252.983,E2 -15252.983} C_VEL
LIN {X 0,Y 319.557,Z 201.49,A -85,B 0,C 180,E1 -15257.016,E2 -15257.016} C_VEL
LIN {X 0,Y 319.549,Z 201.495,A -85,B 0,C 180,E1 -15260.37,E2 -15260.37} C_VEL
LIN {X 0,Y 319.584,Z 201.488,A -85,B 0,C 180,E1 -15264.457,E2 -15264.457} C_VEL
LIN {X 0,Y 319.535,Z 201.497,A -85,B 0,C 180,E1 -15268.138,E2 -15268.138} C_VEL
LIN {X 0,Y 319.615,Z 201.484,A -85,B 0,C 180,E1 -15271.59,E2 -15271.59} C_VEL
LIN {X 0,Y 319.607,Z 201.484,A -85,B 0,C 180,E1 -15275.303,E2 -15275.303} C_VEL
LIN {X 0,Y 319.607,Z 201.485,A -85,B 0,C 180,E1 -15279.4,E2 -15279.4} C_VEL
LIN {X 0,Y 319.663,Z 201.478,A -85,B 0,C 180,E1 -15282.072,E2 -15282.072} C_VEL
LIN {X 0,Y 319.736,Z 201.468,A -85,B 0,C 180,E1 -15286.007,E2 -15286.007} C_VEL
LIN {X 0,Y 319.739,Z 201.468,A -85,B 0,C 180,E1 -15289.871,E2 -15289.871} C_VEL
LIN {X 0,Y 319.939,Z 201.444,A -85,B 0,C 180,E1 -15293.693,E2 -15293.693} C_VEL
LIN {X 0,Y 319.992,Z 201.438,A -85,B 0,C 180,E1 -15297.481,E2 -15297.481} C_VEL
LIN {X 0,Y 320.133,Z 201.417,A -85,B 0,C 180,E1 -15299.999,E2 -15299.999} C_VEL
LIN {X 0,Y 319.992,Z 201.436,A -85,B 0,C 180,E1 -15302.516,E2 -15302.516} C_VEL
LIN {X 0,Y 319.914,Z 201.443,A -85,B 0,C 180,E1 -15306.611,E2 -15306.611} C_VEL
LIN {X 0,Y 319.737,Z 201.467,A -85,B 0,C 180,E1 -15310.127,E2 -15310.127} C_VEL
LIN {X 0,Y 319.733,Z 201.467,A -85,B 0,C 180,E1 -15313.991,E2 -15313.991} C_VEL
LIN {X 0,Y 319.614,Z 201.482,A -85,B 0,C 180,E1 -15317.928,E2 -15317.928} C_VEL
LIN {X 0,Y 319.568,Z 201.488,A -85,B 0,C 180,E1 -15321.953,E2 -15321.953} C_VEL
LIN {X 0,Y 319.634,Z 201.482,A -85,B 0,C 180,E1 -15326.087,E2 -15326.087} C_VEL
LIN {X 0,Y 319.588,Z 201.486,A -85,B 0,C 180,E1 -15328.932,E2 -15328.932} C_VEL
LIN {X 0,Y 319.531,Z 201.494,A -85,B 0,C 180,E1 -15331.86,E2 -15331.86} C_VEL
LIN {X 0,Y 319.577,Z 201.487,A -85,B 0,C 180,E1 -15335.542,E2 -15335.542} C_VEL
LIN {X 0,Y 319.57,Z 201.492,A -85,B 0,C 180,E1 -15338.007,E2 -15338.007} C_VEL
LIN {X 0,Y 319.522,Z 201.495,A -85,B 0,C 180,E1 -15341.596,E2 -15341.596} C_VEL
LIN {X 0,Y 319.484,Z 201.499,A -85,B 0,C 180,E1 -15345.256,E2 -15345.256} C_VEL
LIN {X 0,Y 319.523,Z 201.493,A -85,B 0,C 180,E1 -15348.71,E2 -15348.71} C_VEL
LIN {X 0,Y 319.556,Z 201.49,A -85,B 0,C 180,E1 -15352.347,E2 -15352.347} C_VEL
LIN {X 0,Y 319.554,Z 201.49,A -85,B 0,C 180,E1 -15355.122,E2 -15355.122} C_VEL
LIN {X 0,Y 319.564,Z 201.489,A -85,B 0,C 180,E1 -15359.057,E2 -15359.057} C_VEL
LIN {X 0,Y 319.602,Z 201.483,A -85,B 0,C 180,E1 -15362.497,E2 -15362.497} C_VEL
LIN {X 0,Y 319.598,Z 201.488,A -85,B 0,C 180,E1 -15365.303,E2 -15365.303} C_VEL
LIN {X 0,Y 319.59,Z 201.485,A -85,B 0,C 180,E1 -15368.047,E2 -15368.047} C_VEL
LIN {X 0,Y 319.682,Z 201.476,A -85,B 0,C 180,E1 -15370.961,E2 -15370.961} C_VEL
LIN {X 0,Y 319.723,Z 201.473,A -85,B 0,C 180,E1 -15375.275,E2 -15375.275} C_VEL
LIN {X 0,Y 319.752,Z 201.465,A -85,B 0,C 180,E1 -15379.872,E2 -15379.872} C_VEL
LIN {X 0,Y 319.925,Z 201.444,A -85,B 0,C 180,E1 -15382.426,E2 -15382.426} C_VEL
LIN {X 0,Y 319.739,Z 201.471,A -85,B 0,C 180,E1 -15384.956,E2 -15384.956} C_VEL
LIN {X 0,Y 319.981,Z 201.437,A -85,B 0,C 180,E1 -15387.482,E2 -15387.482} C_VEL
LIN {X 0,Y 320.142,Z 201.417,A -85,B 0,C 180,E1 -15390,E2 -15390} C_VEL
LIN {X 0,Y 319.983,Z 201.44,A -85,B 0,C 180,E1 -15392.517,E2 -15392.517} C_VEL
LIN {X 0,Y 319.944,Z 201.444,A -85,B 0,C 180,E1 -15396.305,E2 -15396.305} C_VEL
LIN {X 0,Y 319.877,Z 201.452,A -85,B 0,C 180,E1 -15398.847,E2 -15398.847} C_VEL
LIN {X 0,Y 319.566,Z 201.491,A -85,B 0,C 180,E1 -15402.704,E2 -15402.704} C_VEL
LIN {X 0,Y 319.264,Z 201.537,A -85,B 0,C 180,E1 -15405.48,E2 -15405.48} C_VEL
LIN {X 0,Y 318.829,Z 205.965,A -85,B 0,C 180,E1 -15409.308,E2 -15409.308} C_VEL
LIN {X 0,Y 318.563,Z 210.815,A -85,B 0,C 180,E1 -15413.397,E2 -15413.397} C_VEL
LIN {X 0,Y 318.381,Z 214.199,A -85,B 0,C 180,E1 -15416.198,E2 -15416.198} C_VEL
LIN {X 0,Y 318.222,Z 218.108,A -85,B 0,C 180,E1 -15419.387,E2 -15419.387} C_VEL
LIN {X 0,Y 319.89,Z 227.719,A -85,B 0,C 180,E1 -15419.988,E2 -15419.988} C_VEL
LIN {X 0,Y 321.218,Z 236.87,A -85,B 0,C 180,E1 -15420.735,E2 -15420.735} C_VEL
LIN {X 0,Y 321.803,Z 242.741,A -85,B 0,C 180,E1 -15421.301,E2 -15421.301} C_VEL
LIN {X 0,Y 321.211,Z 251.012,A -85,B 0,C 180,E1 -15422.23,E2 -15422.23} C_VEL
LIN {X 0,Y 320.634,Z 258.253,A -85,B 0,C 180,E1 -15423.228,E2 -15423.228} C_VEL
LIN {X 0,Y 320.1,Z 263.918,A -85,B 0,C 180,E1 -15424.158,E2 -15424.158} C_VEL
LIN {X 0,Y 319.629,Z 269.209,A -85,B 0,C 180,E1 -15425.182,E2 -15425.182} C_VEL
LIN {X 0,Y 319.175,Z 274.759,A -85,B 0,C 180,E1 -15426.478,E2 -15426.478} C_VEL
LIN {X 0,Y 318.624,Z 280.461,A -85,B 0,C 180,E1 -15428.141,E2 -15428.141} C_VEL
LIN {X 0,Y 318.188,Z 284.928,A -85,B 0,C 180,E1 -15429.832,E2 -15429.832} C_VEL
LIN {X 0,Y 317.924,Z 288.192,A -85,B 0,C 180,E1 -15431.543,E2 -15431.543} C_VEL
LIN {X 0,Y 317.758,Z 290.345,A -85,B 0,C 180,E1 -15433.286,E2 -15433.286} C_VEL
LIN {X 0,Y 317.72,Z 291.475,A -85,B 0,C 180,E1 -15435.059,E2 -15435.059} C_VEL
LIN {X 0,Y 317.8,Z 291.565,A -85,B 0,C 180,E1 -15436.868,E2 -15436.868} C_VEL
LIN {X 0,Y 318.108,Z 290.571,A -85,B 0,C 180,E1 -15438.691,E2 -15438.691} C_VEL
LIN {X 0,Y 318.56,Z 288.394,A -85,B 0,C 180,E1 -15440.548,E2 -15440.548} C_VEL
LIN {X 0,Y 319.145,Z 284.759,A -85,B 0,C 180,E1 -15442.445,E2 -15442.445} C_VEL
LIN {X 0,Y 319.834,Z 280.634,A -85,B 0,C 180,E1 -15444.021,E2 -15444.021} C_VEL
LIN {X 0,Y 320.597,Z 275.599,A -85,B 0,C 180,E1 -15445.525,E2 -15445.525} C_VEL
LIN {X 0,Y 321.728,Z 268.244,A -85,B 0,C 180,E1 -15447.238,E2 -15447.238} C_VEL
LIN {X 0,Y 322.657,Z 261.351,A -85,B 0,C 180,E1 -15448.484,E2 -15448.484} C_VEL
LIN {X 0,Y 323.55,Z 254.582,A -85,B 0,C 180,E1 -15449.488,E2 -15449.488} C_VEL
LIN {X 0,Y 324.359,Z 246.825,A -85,B 0,C 180,E1 -15450.435,E2 -15450.435} C_VEL
LIN {X 0,Y 323.487,Z 239.501,A -85,B 0,C 180,E1 -15451.272,E2 -15451.272} C_VEL
LIN {X 0,Y 321.716,Z 230.763,A -85,B 0,C 180,E1 -15452.139,E2 -15452.139} C_VEL
LIN {X 0,Y 318.723,Z 219.522,A -85,B 0,C 180,E1 -15453.083,E2 -15453.083} C_VEL
LIN {X 0,Y 318.984,Z 215.646,A -85,B 0,C 180,E1 -15456.637,E2 -15456.637} C_VEL
LIN {X 0,Y 319.357,Z 211.62,A -85,B 0,C 180,E1 -15460.464,E2 -15460.464} C_VEL
LIN {X 0,Y 318.85,Z 210.651,A -85,B 0,C 180,E1 -15461.503,E2 -15461.503} C_VEL
LIN {X 0,Y 316.246,Z 209.38,A -85,B 0,C 180,E1 -15463.211,E2 -15463.211} C_VEL
LIN {X 0,Y 313.973,Z 208.429,A -85,B 0,C 180,E1 -15464.596,E2 -15464.596} C_VEL
LIN {X 0,Y 312.994,Z 207.595,A -85,B 0,C 180,E1 -15465.662,E2 -15465.662} C_VEL
LIN {X 0,Y 312.915,Z 207.275,A -85,B 0,C 180,E1 -15466.021,E2 -15466.021} C_VEL
LIN {X 0,Y 312.984,Z 205.185,A -85,B 0,C 180,E1 -15468.342,E2 -15468.342} C_VEL
LIN {X 0,Y 312.862,Z 202.665,A -85,B 0,C 180,E1 -15471.263,E2 -15471.263} C_VEL
LIN {X 0,Y 312.911,Z 202.329,A -85,B 0,C 180,E1 -15473.553,E2 -15473.553} C_VEL
LIN {X 0,Y 312.937,Z 202.32,A -85,B 0,C 180,E1 -15477.427,E2 -15477.427} C_VEL
LIN {X 0,Y 313.121,Z 202.295,A -85,B 0,C 180,E1 -15480.001,E2 -15480.001} C_VEL
LIN {X 0,Y 312.937,Z 202.317,A -85,B 0,C 180,E1 -15482.575,E2 -15482.575} C_VEL
LIN {X 0,Y 312.895,Z 202.323,A -85,B 0,C 180,E1 -15486.449,E2 -15486.449} C_VEL
LIN {X 0,Y 312.687,Z 202.349,A -85,B 0,C 180,E1 -15490.36,E2 -15490.36} C_VEL
LIN {X 0,Y 312.702,Z 202.347,A -85,B 0,C 180,E1 -15494.889,E2 -15494.889} C_VEL
LIN {X 0,Y 312.634,Z 202.355,A -85,B 0,C 180,E1 -15499.238,E2 -15499.238} C_VEL
LIN {X 0,Y 312.548,Z 202.367,A -85,B 0,C 180,E1 -15502.79,E2 -15502.79} C_VEL
LIN {X 0,Y 312.605,Z 202.356,A -85,B 0,C 180,E1 -15505.936,E2 -15505.936} C_VEL
LIN {X 0,Y 312.547,Z 202.367,A -85,B 0,C 180,E1 -15509.651,E2 -15509.651} C_VEL
LIN {X 0,Y 312.522,Z 202.368,A -85,B 0,C 180,E1 -15513.689,E2 -15513.689} C_VEL
LIN {X 0,Y 312.528,Z 202.369,A -85,B 0,C 180,E1 -15517.386,E2 -15517.386} C_VEL
LIN {X 0,Y 312.492,Z 202.376,A -85,B 0,C 180,E1 -15520.71,E2 -15520.71} C_VEL
LIN {X 0,Y 312.454,Z 202.383,A -85,B 0,C 180,E1 -15524.21,E2 -15524.21} C_VEL
LIN {X 0,Y 312.476,Z 202.501,A -85,B 0,C 180,E1 -15525.542,E2 -15525.542} C_VEL
LIN {X 0,Y 313.306,Z 206.728,A -85,B 0,C 180,E1 -15529.419,E2 -15529.419} C_VEL
LIN {X 0,Y 314.134,Z 210.912,A -85,B 0,C 180,E1 -15532.839,E2 -15532.839} C_VEL
LIN {X 0,Y 315.058,Z 216.405,A -85,B 0,C 180,E1 -15536.871,E2 -15536.871} C_VEL
LIN {X 0,Y 315.156,Z 217.986,A -85,B 0,C 180,E1 -15537.931,E2 -15537.931} C_VEL
LIN {X 0,Y 314.402,Z 222.335,A -85,B 0,C 180,E1 -15540.668,E2 -15540.668} C_VEL
LIN {X 0,Y 313.199,Z 229.219,A -85,B 0,C 180,E1 -15544.764,E2 -15544.764} C_VEL
LIN {X 0,Y 312.24,Z 236.455,A -85,B 0,C 180,E1 -15548.892,E2 -15548.892} C_VEL
LIN {X 0,Y 311.923,Z 239.417,A -85,B 0,C 180,E1 -15550.544,E2 -15550.544} C_VEL
LIN {X 0,Y 314.481,Z 252.464,A -85,B 0,C 180,E1 -15551.481,E2 -15551.481} C_VEL
LIN {X 0,Y 315.606,Z 262.07,A -85,B 0,C 180,E1 -15552.338,E2 -15552.338} C_VEL
LIN {X 0,Y 316.046,Z 270.233,A -85,B 0,C 180,E1 -15553.197,E2 -15553.197} C_VEL
LIN {X 0,Y 315.982,Z 277.448,A -85,B 0,C 180,E1 -15554.081,E2 -15554.081} C_VEL
LIN {X 0,Y 315.069,Z 284.941,A -85,B 0,C 180,E1 -15555.136,E2 -15555.136} C_VEL
LIN {X 0,Y 314.216,Z 290.665,A -85,B 0,C 180,E1 -15556.088,E2 -15556.088} C_VEL
LIN {X 0,Y 313.292,Z 297.07,A -85,B 0,C 180,E1 -15557.366,E2 -15557.366} C_VEL
LIN {X 0,Y 312.36,Z 303.593,A -85,B 0,C 180,E1 -15558.975,E2 -15558.975} C_VEL
LIN {X 0,Y 311.797,Z 307.847,A -85,B 0,C 180,E1 -15560.268,E2 -15560.268} C_VEL
LIN {X 0,Y 311.335,Z 311.38,A -85,B 0,C 180,E1 -15561.563,E2 -15561.563} C_VEL
LIN {X 0,Y 310.906,Z 315.464,A -85,B 0,C 180,E1 -15563.511,E2 -15563.511} C_VEL
LIN {X 0,Y 310.777,Z 317.453,A -85,B 0,C 180,E1 -15564.81,E2 -15564.81} C_VEL
LIN {X 0,Y 310.777,Z 318.928,A -85,B 0,C 180,E1 -15566.11,E2 -15566.11} C_VEL
LIN {X 0,Y 310.743,Z 319.901,A -85,B 0,C 180,E1 -15567.408,E2 -15567.408} C_VEL
LIN {X 0,Y 310.774,Z 320.291,A -85,B 0,C 180,E1 -15568.704,E2 -15568.704} C_VEL
LIN {X 0,Y 310.858,Z 320.144,A -85,B 0,C 180,E1 -15570,E2 -15570} C_VEL
LIN {X 0,Y 310.813,Z 319.507,A -85,B 0,C 180,E1 -15571.296,E2 -15571.296} C_VEL
LIN {X 0,Y 310.766,Z 318.371,A -85,B 0,C 180,E1 -15572.593,E2 -15572.593} C_VEL
LIN {X 0,Y 310.869,Z 316.716,A -85,B 0,C 180,E1 -15573.889,E2 -15573.889} C_VEL
LIN {X 0,Y 310.84,Z 313.018,A -85,B 0,C 180,E1 -15575.825,E2 -15575.825} C_VEL
LIN {X 0,Y 311.132,Z 307.845,A -85,B 0,C 180,E1 -15577.79,E2 -15577.79} C_VEL
LIN {X 0,Y 311.536,Z 302.288,A -85,B 0,C 180,E1 -15579.414,E2 -15579.414} C_VEL
LIN {X 0,Y 312.106,Z 295.239,A -85,B 0,C 180,E1 -15581.035,E2 -15581.035} C_VEL
LIN {X 0,Y 312.825,Z 287.154,A -85,B 0,C 180,E1 -15582.488,E2 -15582.488} C_VEL
LIN {X 0,Y 313.47,Z 280.658,A -85,B 0,C 180,E1 -15583.451,E2 -15583.451} C_VEL
LIN {X 0,Y 313.98,Z 273.113,A -85,B 0,C 180,E1 -15584.382,E2 -15584.382} C_VEL
LIN {X 0,Y 313.549,Z 265.165,A -85,B 0,C 180,E1 -15585.208,E2 -15585.208} C_VEL
LIN {X 0,Y 312.864,Z 256.006,A -85,B 0,C 180,E1 -15585.973,E2 -15585.973} C_VEL
LIN {X 0,Y 311.846,Z 245.58,A -85,B 0,C 180,E1 -15586.636,E2 -15586.636} C_VEL
LIN {X 0,Y 311.354,Z 240.707,A -85,B 0,C 180,E1 -15586.895,E2 -15586.895} C_VEL
LIN {X 0,Y 311.834,Z 234.126,A -85,B 0,C 180,E1 -15590.447,E2 -15590.447} C_VEL
LIN {X 0,Y 312.483,Z 227.82,A -85,B 0,C 180,E1 -15593.881,E2 -15593.881} C_VEL
LIN {X 0,Y 313.322,Z 221.51,A -85,B 0,C 180,E1 -15597.376,E2 -15597.376} C_VEL
LIN {X 0,Y 314.261,Z 215.153,A -85,B 0,C 180,E1 -15600.955,E2 -15600.955} C_VEL
LIN {X 0,Y 314.358,Z 212.604,A -85,B 0,C 180,E1 -15602.45,E2 -15602.45} C_VEL
LIN {X 0,Y 313.492,Z 207.404,A -85,B 0,C 180,E1 -15605.654,E2 -15605.654} C_VEL
LIN {X 0,Y 312.583,Z 202.366,A -85,B 0,C 180,E1 -15609.017,E2 -15609.017} C_VEL
LIN {X 0,Y 312.494,Z 202.374,A -85,B 0,C 180,E1 -15612.431,E2 -15612.431} C_VEL
LIN {X 0,Y 312.462,Z 202.375,A -85,B 0,C 180,E1 -15616.035,E2 -15616.035} C_VEL
LIN {X 0,Y 312.508,Z 202.369,A -85,B 0,C 180,E1 -15619.874,E2 -15619.874} C_VEL
LIN {X 0,Y 312.539,Z 202.368,A -85,B 0,C 180,E1 -15624.05,E2 -15624.05} C_VEL
LIN {X 0,Y 312.508,Z 202.368,A -85,B 0,C 180,E1 -15627.333,E2 -15627.333} C_VEL
LIN {X 0,Y 312.548,Z 202.363,A -85,B 0,C 180,E1 -15631.278,E2 -15631.278} C_VEL
LIN {X 0,Y 312.589,Z 202.357,A -85,B 0,C 180,E1 -15634.71,E2 -15634.71} C_VEL
LIN {X 0,Y 312.542,Z 202.363,A -85,B 0,C 180,E1 -15638.912,E2 -15638.912} C_VEL
LIN {X 0,Y 312.643,Z 202.356,A -85,B 0,C 180,E1 -15641.656,E2 -15641.656} C_VEL
LIN {X 0,Y 312.698,Z 202.348,A -85,B 0,C 180,E1 -15645.685,E2 -15645.685} C_VEL
LIN {X 0,Y 312.69,Z 202.348,A -85,B 0,C 180,E1 -15649.64,E2 -15649.64} C_VEL
LIN {X 0,Y 312.896,Z 202.323,A -85,B 0,C 180,E1 -15653.551,E2 -15653.551} C_VEL
LIN {X 0,Y 312.938,Z 202.317,A -85,B 0,C 180,E1 -15657.425,E2 -15657.425} C_VEL
LIN {X 0,Y 313.086,Z 202.295,A -85,B 0,C 180,E1 -15659.999,E2 -15659.999} C_VEL
LIN {X 0,Y 312.938,Z 202.315,A -85,B 0,C 180,E1 -15662.573,E2 -15662.573} C_VEL
LIN {X 0,Y 312.88,Z 202.321,A -85,B 0,C 180,E1 -15666.589,E2 -15666.589} C_VEL
LIN {X 0,Y 312.687,Z 202.346,A -85,B 0,C 180,E1 -15670.357,E2 -15670.357} C_VEL
LIN {X 0,Y 312.669,Z 202.352,A -85,B 0,C 180,E1 -15674.864,E2 -15674.864} C_VEL
LIN {X 0,Y 312.549,Z 202.363,A -85,B 0,C 180,E1 -15679.192,E2 -15679.192} C_VEL
LIN {X 0,Y 312.526,Z 202.368,A -85,B 0,C 180,E1 -15682.779,E2 -15682.779} C_VEL
LIN {X 0,Y 312.602,Z 202.357,A -85,B 0,C 180,E1 -15685.934,E2 -15685.934} C_VEL
LIN {X 0,Y 312.544,Z 202.363,A -85,B 0,C 180,E1 -15689.648,E2 -15689.648} C_VEL
LIN {X 0,Y 312.517,Z 202.367,A -85,B 0,C 180,E1 -15693.687,E2 -15693.687} C_VEL
LIN {X 0,Y 312.534,Z 202.364,A -85,B 0,C 180,E1 -15697.382,E2 -15697.382} C_VEL
LIN {X 0,Y 312.486,Z 202.37,A -85,B 0,C 180,E1 -15700.708,E2 -15700.708} C_VEL
LIN {X 0,Y 312.447,Z 202.378,A -85,B 0,C 180,E1 -15704.208,E2 -15704.208} C_VEL
LIN {X 0,Y 312.479,Z 202.376,A -85,B 0,C 180,E1 -15707.917,E2 -15707.917} C_VEL
LIN {X 0,Y 312.529,Z 202.369,A -85,B 0,C 180,E1 -15711.909,E2 -15711.909} C_VEL
LIN {X 0,Y 312.501,Z 202.372,A -85,B 0,C 180,E1 -15715.789,E2 -15715.789} C_VEL
LIN {X 0,Y 312.518,Z 202.366,A -85,B 0,C 180,E1 -15718.853,E2 -15718.853} C_VEL
LIN {X 0,Y 312.576,Z 202.361,A -85,B 0,C 180,E1 -15721.825,E2 -15721.825} C_VEL
LIN {X 0,Y 312.579,Z 202.359,A -85,B 0,C 180,E1 -15724.71,E2 -15724.71} C_VEL
LIN {X 0,Y 312.58,Z 202.362,A -85,B 0,C 180,E1 -15727.528,E2 -15727.528} C_VEL
LIN {X 0,Y 312.631,Z 202.354,A -85,B 0,C 180,E1 -15731.656,E2 -15731.656} C_VEL
LIN {X 0,Y 312.686,Z 202.346,A -85,B 0,C 180,E1 -15735.686,E2 -15735.686} C_VEL
LIN {X 0,Y 312.696,Z 202.345,A -85,B 0,C 180,E1 -15739.641,E2 -15739.641} C_VEL
LIN {X 0,Y 312.864,Z 202.323,A -85,B 0,C 180,E1 -15742.254,E2 -15742.254} C_VEL
LIN {X 0,Y 312.709,Z 202.347,A -85,B 0,C 180,E1 -15744.842,E2 -15744.842} C_VEL
LIN {X 0,Y 312.984,Z 202.313,A -85,B 0,C 180,E1 -15748.713,E2 -15748.713} C_VEL
LIN {X 0,Y 312.982,Z 202.309,A -85,B 0,C 180,E1 -15751.286,E2 -15751.286} C_VEL
LIN {X 0,Y 312.71,Z 202.343,A -85,B 0,C 180,E1 -15755.158,E2 -15755.158} C_VEL
LIN {X 0,Y 312.875,Z 202.321,A -85,B 0,C 180,E1 -15757.745,E2 -15757.745} C_VEL
LIN {X 0,Y 312.667,Z 202.352,A -85,B 0,C 180,E1 -15760.359,E2 -15760.359} C_VEL
LIN {X 0,Y 312.403,Z 202.386,A -85,B 0,C 180,E1 -15764.327,E2 -15764.327} C_VEL
LIN {X 0,Y 312.153,Z 202.614,A -85,B 0,C 180,E1 -15765.674,E2 -15765.674} C_VEL
LIN {X 0,Y 311.721,Z 207.28,A -85,B 0,C 180,E1 -15769.766,E2 -15769.766} C_VEL
LIN {X 0,Y 311.488,Z 212.184,A -85,B 0,C 180,E1 -15773.962,E2 -15773.962} C_VEL
LIN {X 0,Y 311.191,Z 217.326,A -85,B 0,C 180,E1 -15778.266,E2 -15778.266} C_VEL
LIN {X 0,Y 311.174,Z 218.333,A -85,B 0,C 180,E1 -15779.097,E2 -15779.097} C_VEL
LIN {X 0,Y 312.958,Z 228.886,A -85,B 0,C 180,E1 -15779.792,E2 -15779.792} C_VEL
LIN {X 0,Y 314.292,Z 238.086,A -85,B 0,C 180,E1 -15780.579,E2 -15780.579} C_VEL
LIN {X 0,Y 314.821,Z 242.908,A -85,B 0,C 180,E1 -15781.06,E2 -15781.06} C_VEL
LIN {X 0,Y 314.158,Z 252.022,A -85,B 0,C 180,E1 -15782.116,E2 -15782.116} C_VEL
LIN {X 0,Y 313.486,Z 260.288,A -85,B 0,C 180,E1 -15783.316,E2 -15783.316} C_VEL
LIN {X 0,Y 312.699,Z 268.303,A -85,B 0,C 180,E1 -15784.772,E2 -15784.772} C_VEL
LIN {X 0,Y 312.183,Z 274.54,A -85,B 0,C 180,E1 -15786.224,E2 -15786.224} C_VEL
LIN {X 0,Y 311.605,Z 280.191,A -85,B 0,C 180,E1 -15787.873,E2 -15787.873} C_VEL
LIN {X 0,Y 311.224,Z 283.857,A -85,B 0,C 180,E1 -15789.219,E2 -15789.219} C_VEL
LIN {X 0,Y 310.913,Z 287.491,A -85,B 0,C 180,E1 -15790.959,E2 -15790.959} C_VEL
LIN {X 0,Y 310.707,Z 290.073,A -85,B 0,C 180,E1 -15792.733,E2 -15792.733} C_VEL
LIN {X 0,Y 310.643,Z 291.603,A -85,B 0,C 180,E1 -15794.535,E2 -15794.535} C_VEL
LIN {X 0,Y 310.687,Z 292.028,A -85,B 0,C 180,E1 -15796.375,E2 -15796.375} C_VEL
LIN {X 0,Y 310.934,Z 291.357,A -85,B 0,C 180,E1 -15798.236,E2 -15798.236} C_VEL
LIN {X 0,Y 311.101,Z 290.767,A -85,B 0,C 180,E1 -15799.072,E2 -15799.072} C_VEL
LIN {X 0,Y 311.565,Z 288.64,A -85,B 0,C 180,E1 -15800.834,E2 -15800.834} C_VEL
LIN {X 0,Y 312.106,Z 285.458,A -85,B 0,C 180,E1 -15802.558,E2 -15802.558} C_VEL
LIN {X 0,Y 312.87,Z 281.143,A -85,B 0,C 180,E1 -15804.267,E2 -15804.267} C_VEL
LIN {X 0,Y 313.531,Z 277.121,A -85,B 0,C 180,E1 -15805.53,E2 -15805.53} C_VEL
LIN {X 0,Y 314.317,Z 272.229,A -85,B 0,C 180,E1 -15806.793,E2 -15806.793} C_VEL
LIN {X 0,Y 315.318,Z 265.596,A -85,B 0,C 180,E1 -15808.185,E2 -15808.185} C_VEL
LIN {X 0,Y 316.467,Z 258.027,A -85,B 0,C 180,E1 -15809.461,E2 -15809.461} C_VEL
LIN {X 0,Y 317.523,Z 248.564,A -85,B 0,C 180,E1 -15810.721,E2 -15810.721} C_VEL
LIN {X 0,Y 316.948,Z 241.927,A -85,B 0,C 180,E1 -15811.529,E2 -15811.529} C_VEL
LIN {X 0,Y 315.314,Z 233.273,A -85,B 0,C 180,E1 -15812.453,E2 -15812.453} C_VEL
LIN {X 0,Y 312.862,Z 223.983,A -85,B 0,C 180,E1 -15813.305,E2 -15813.305} C_VEL
LIN {X 0,Y 311.708,Z 219.829,A -85,B 0,C 180,E1 -15813.65,E2 -15813.65} C_VEL
LIN {X 0,Y 312.051,Z 215.762,A -85,B 0,C 180,E1 -15817.49,E2 -15817.49} C_VEL
LIN {X 0,Y 312.483,Z 211.513,A -85,B 0,C 180,E1 -15821.648,E2 -15821.648} C_VEL
LIN {X 0,Y 312.922,Z 207.568,A -85,B 0,C 180,E1 -15825.698,E2 -15825.698} C_VEL
LIN {X 0,Y 312.915,Z 207.275,A -85,B 0,C 180,E1 -15826.021,E2 -15826.021} C_VEL
LIN {X 0,Y 312.252,Z 206.439,A -85,B 0,C 180,E1 -15827.085,E2 -15827.085} C_VEL
LIN {X 0,Y 309.408,Z 205.407,A -85,B 0,C 180,E1 -15828.825,E2 -15828.825} C_VEL
LIN {X 0,Y 306.988,Z 204.654,A -85,B 0,C 180,E1 -15830.238,E2 -15830.238} C_VEL
LIN {X 0,Y 305.938,Z 203.958,A -85,B 0,C 180,E1 -15831.329,E2 -15831.329} C_VEL
LIN {X 0,Y 305.847,Z 203.681,A -85,B 0,C 180,E1 -15831.698,E2 -15831.698} C_VEL
LIN {X 0,Y 305.853,Z 203.207,A -85,B 0,C 180,E1 -15833.404,E2 -15833.404} C_VEL
LIN {X 0,Y 305.958,Z 203.188,A -85,B 0,C 180,E1 -15838.685,E2 -15838.685} C_VEL
LIN {X 0,Y 305.958,Z 203.185,A -85,B 0,C 180,E1 -15841.317,E2 -15841.317} C_VEL
LIN {X 0,Y 305.686,Z 203.221,A -85,B 0,C 180,E1 -15845.278,E2 -15845.278} C_VEL
LIN {X 0,Y 305.773,Z 203.21,A -85,B 0,C 180,E1 -15847.928,E2 -15847.928} C_VEL
LIN {X 0,Y 305.601,Z 203.232,A -85,B 0,C 180,E1 -15851.946,E2 -15851.946} C_VEL
LIN {X 0,Y 305.64,Z 203.227,A -85,B 0,C 180,E1 -15855.036,E2 -15855.036} C_VEL
LIN {X 0,Y 305.58,Z 203.234,A -85,B 0,C 180,E1 -15859.446,E2 -15859.446} C_VEL
LIN {X 0,Y 305.493,Z 203.245,A -85,B 0,C 180,E1 -15863.042,E2 -15863.042} C_VEL
LIN {X 0,Y 305.55,Z 203.236,A -85,B 0,C 180,E1 -15866.228,E2 -15866.228} C_VEL
LIN {X 0,Y 305.498,Z 203.244,A -85,B 0,C 180,E1 -15869.051,E2 -15869.051} C_VEL
LIN {X 0,Y 305.446,Z 203.25,A -85,B 0,C 180,E1 -15871.953,E2 -15871.953} C_VEL
LIN {X 0,Y 305.465,Z 203.247,A -85,B 0,C 180,E1 -15875.114,E2 -15875.114} C_VEL
LIN {X 0,Y 305.469,Z 203.249,A -85,B 0,C 180,E1 -15878.533,E2 -15878.533} C_VEL
LIN {X 0,Y 305.457,Z 203.253,A -85,B 0,C 180,E1 -15882.586,E2 -15882.586} C_VEL
LIN {X 0,Y 305.404,Z 203.328,A -85,B 0,C 180,E1 -15884.663,E2 -15884.663} C_VEL
LIN {X 0,Y 306.114,Z 207.016,A -85,B 0,C 180,E1 -15888.256,E2 -15888.256} C_VEL
LIN {X 0,Y 306.957,Z 211.134,A -85,B 0,C 180,E1 -15891.817,E2 -15891.817} C_VEL
LIN {X 0,Y 307.745,Z 215.616,A -85,B 0,C 180,E1 -15895.3,E2 -15895.3} C_VEL
LIN {X 0,Y 308.212,Z 218.687,A -85,B 0,C 180,E1 -15897.533,E2 -15897.533} C_VEL
LIN {X 0,Y 307.512,Z 222.921,A -85,B 0,C 180,E1 -15900.282,E2 -15900.282} C_VEL
LIN {X 0,Y 306.138,Z 230.411,A -85,B 0,C 180,E1 -15904.868,E2 -15904.868} C_VEL
LIN {X 0,Y 305.13,Z 237.602,A -85,B 0,C 180,E1 -15909.084,E2 -15909.084} C_VEL
LIN {X 0,Y 304.955,Z 239.097,A -85,B 0,C 180,E1 -15909.936,E2 -15909.936} C_VEL
LIN {X 0,Y 307.507,Z 251.705,A -85,B 0,C 180,E1 -15910.882,E2 -15910.882} C_VEL
LIN {X 0,Y 308.729,Z 261.22,A -85,B 0,C 180,E1 -15911.76,E2 -15911.76} C_VEL
LIN {X 0,Y 309.229,Z 269.549,A -85,B 0,C 180,E1 -15912.662,E2 -15912.662} C_VEL
LIN {X 0,Y 309.157,Z 277.917,A -85,B 0,C 180,E1 -15913.729,E2 -15913.729} C_VEL
LIN {X 0,Y 308.24,Z 285.217,A -85,B 0,C 180,E1 -15914.799,E2 -15914.799} C_VEL
LIN {X 0,Y 307.077,Z 292.546,A -85,B 0,C 180,E1 -15916.095,E2 -15916.095} C_VEL
LIN {X 0,Y 305.976,Z 300.007,A -85,B 0,C 180,E1 -15917.733,E2 -15917.733} C_VEL
LIN {X 0,Y 305.051,Z 305.869,A -85,B 0,C 180,E1 -15919.379,E2 -15919.379} C_VEL
LIN {X 0,Y 304.533,Z 309.712,A -85,B 0,C 180,E1 -15920.704,E2 -15920.704} C_VEL
LIN {X 0,Y 303.964,Z 314.125,A -85,B 0,C 180,E1 -15922.694,E2 -15922.694} C_VEL
LIN {X 0,Y 303.688,Z 317.244,A -85,B 0,C 180,E1 -15924.689,E2 -15924.689} C_VEL
LIN {X 0,Y 303.688,Z 318.668,A -85,B 0,C 180,E1 -15926.019,E2 -15926.019} C_VEL
LIN {X 0,Y 303.666,Z 319.6,A -85,B 0,C 180,E1 -15927.347,E2 -15927.347} C_VEL
LIN {X 0,Y 303.684,Z 319.981,A -85,B 0,C 180,E1 -15928.674,E2 -15928.674} C_VEL
LIN {X 0,Y 303.766,Z 319.791,A -85,B 0,C 180,E1 -15930,E2 -15930} C_VEL
LIN {X 0,Y 303.721,Z 319.11,A -85,B 0,C 180,E1 -15931.326,E2 -15931.326} C_VEL
LIN {X 0,Y 303.691,Z 317.927,A -85,B 0,C 180,E1 -15932.653,E2 -15932.653} C_VEL
LIN {X 0,Y 303.777,Z 316.228,A -85,B 0,C 180,E1 -15933.98,E2 -15933.98} C_VEL
LIN {X 0,Y 303.739,Z 312.936,A -85,B 0,C 180,E1 -15935.757,E2 -15935.757} C_VEL
LIN {X 0,Y 303.961,Z 309.157,A -85,B 0,C 180,E1 -15937.306,E2 -15937.306} C_VEL
LIN {X 0,Y 304.303,Z 303.967,A -85,B 0,C 180,E1 -15938.969,E2 -15938.969} C_VEL
LIN {X 0,Y 304.706,Z 298.864,A -85,B 0,C 180,E1 -15940.297,E2 -15940.297} C_VEL
LIN {X 0,Y 305.252,Z 292.702,A -85,B 0,C 180,E1 -15941.622,E2 -15941.622} C_VEL
LIN {X 0,Y 305.865,Z 286.218,A -85,B 0,C 180,E1 -15942.777,E2 -15942.777} C_VEL
LIN {X 0,Y 306.597,Z 278.368,A -85,B 0,C 180,E1 -15943.927,E2 -15943.927} C_VEL
LIN {X 0,Y 306.898,Z 273.018,A -85,B 0,C 180,E1 -15944.59,E2 -15944.59} C_VEL
LIN {X 0,Y 306.474,Z 264.631,A -85,B 0,C 180,E1 -15945.482,E2 -15945.482} C_VEL
LIN {X 0,Y 305.739,Z 255.384,A -85,B 0,C 180,E1 -15946.27,E2 -15946.27} C_VEL
LIN {X 0,Y 304.817,Z 245.247,A -85,B 0,C 180,E1 -15946.923,E2 -15946.923} C_VEL
LIN {X 0,Y 304.303,Z 240.404,A -85,B 0,C 180,E1 -15947.212,E2 -15947.212} C_VEL
LIN {X 0,Y 304.999,Z 232.441,A -85,B 0,C 180,E1 -15951.635,E2 -15951.635} C_VEL
LIN {X 0,Y 305.876,Z 224.883,A -85,B 0,C 180,E1 -15955.885,E2 -15955.885} C_VEL
LIN {X 0,Y 306.785,Z 218.6,A -85,B 0,C 180,E1 -15959.479,E2 -15959.479} C_VEL
LIN {X 0,Y 307.342,Z 213.969,A -85,B 0,C 180,E1 -15962.211,E2 -15962.211} C_VEL
LIN {X 0,Y 306.683,Z 209.597,A -85,B 0,C 180,E1 -15964.953,E2 -15964.953} C_VEL
LIN {X 0,Y 305.548,Z 203.288,A -85,B 0,C 180,E1 -15969.081,E2 -15969.081} C_VEL
LIN {X 0,Y 305.459,Z 203.25,A -85,B 0,C 180,E1 -15972.586,E2 -15972.586} C_VEL
LIN {X 0,Y 305.427,Z 203.254,A -85,B 0,C 180,E1 -15976.344,E2 -15976.344} C_VEL
LIN {X 0,Y 305.461,Z 203.247,A -85,B 0,C 180,E1 -15979.892,E2 -15979.892} C_VEL
LIN {X 0,Y 305.467,Z 203.245,A -85,B 0,C 180,E1 -15983.636,E2 -15983.636} C_VEL
LIN {X 0,Y 305.469,Z 203.246,A -85,B 0,C 180,E1 -15986.483,E2 -15986.483} C_VEL
LIN {X 0,Y 305.463,Z 203.247,A -85,B 0,C 180,E1 -15989.59,E2 -15989.59} C_VEL
LIN {X 0,Y 305.523,Z 203.237,A -85,B 0,C 180,E1 -15992.608,E2 -15992.608} C_VEL
LIN {X 0,Y 305.509,Z 203.242,A -85,B 0,C 180,E1 -15995.538,E2 -15995.538} C_VEL
LIN {X 0,Y 305.511,Z 203.243,A -85,B 0,C 180,E1 -15999.813,E2 -15999.813} C_VEL
LIN {X 0,Y 305.579,Z 203.23,A -85,B 0,C 180,E1 -16002.602,E2 -16002.602} C_VEL
LIN {X 0,Y 305.653,Z 203.224,A -85,B 0,C 180,E1 -16005.348,E2 -16005.348} C_VEL
LIN {X 0,Y 305.629,Z 203.229,A -85,B 0,C 180,E1 -16009.398,E2 -16009.398} C_VEL
LIN {X 0,Y 305.775,Z 203.206,A -85,B 0,C 180,E1 -16012.072,E2 -16012.072} C_VEL
LIN {X 0,Y 305.686,Z 203.218,A -85,B 0,C 180,E1 -16014.722,E2 -16014.722} C_VEL
LIN {X 0,Y 305.959,Z 203.184,A -85,B 0,C 180,E1 -16018.683,E2 -16018.683} C_VEL
LIN {X 0,Y 305.957,Z 203.187,A -85,B 0,C 180,E1 -16021.315,E2 -16021.315} C_VEL
LIN {X 0,Y 305.686,Z 203.22,A -85,B 0,C 180,E1 -16025.275,E2 -16025.275} C_VEL
LIN {X 0,Y 305.773,Z 203.206,A -85,B 0,C 180,E1 -16027.925,E2 -16027.925} C_VEL
LIN {X 0,Y 305.601,Z 203.228,A -85,B 0,C 180,E1 -16031.944,E2 -16031.944} C_VEL
LIN {X 0,Y 305.61,Z 203.229,A -85,B 0,C 180,E1 -16035.013,E2 -16035.013} C_VEL
LIN {X 0,Y 305.518,Z 203.242,A -85,B 0,C 180,E1 -16038.786,E2 -16038.786} C_VEL
LIN {X 0,Y 305.486,Z 203.243,A -85,B 0,C 180,E1 -16043.038,E2 -16043.038} C_VEL
LIN {X 0,Y 305.547,Z 203.237,A -85,B 0,C 180,E1 -16046.226,E2 -16046.226} C_VEL
LIN {X 0,Y 305.494,Z 203.242,A -85,B 0,C 180,E1 -16049.048,E2 -16049.048} C_VEL
LIN {X 0,Y 305.443,Z 203.249,A -85,B 0,C 180,E1 -16051.951,E2 -16051.951} C_VEL
LIN {X 0,Y 305.46,Z 203.245,A -85,B 0,C 180,E1 -16055.112,E2 -16055.112} C_VEL
LIN {X 0,Y 305.464,Z 203.246,A -85,B 0,C 180,E1 -16058.531,E2 -16058.531} C_VEL
LIN {X 0,Y 305.451,Z 203.247,A -85,B 0,C 180,E1 -16062.584,E2 -16062.584} C_VEL
LIN {X 0,Y 305.421,Z 203.252,A -85,B 0,C 180,E1 -16066.344,E2 -16066.344} C_VEL
LIN {X 0,Y 305.453,Z 203.251,A -85,B 0,C 180,E1 -16069.891,E2 -16069.891} C_VEL
LIN {X 0,Y 305.476,Z 203.248,A -85,B 0,C 180,E1 -16073.63,E2 -16073.63} C_VEL
LIN {X 0,Y 305.459,Z 203.245,A -85,B 0,C 180,E1 -16076.482,E2 -16076.482} C_VEL
LIN {X 0,Y 305.497,Z 203.242,A -85,B 0,C 180,E1 -16080.946,E2 -16080.946} C_VEL
LIN {X 0,Y 305.566,Z 203.232,A -85,B 0,C 180,E1 -16084.087,E2 -16084.087} C_VEL
LIN {X 0,Y 305.493,Z 203.241,A -85,B 0,C 180,E1 -16088.402,E2 -16088.402} C_VEL
LIN {X 0,Y 305.583,Z 203.235,A -85,B 0,C 180,E1 -16091.217,E2 -16091.217} C_VEL
LIN {X 0,Y 305.641,Z 203.226,A -85,B 0,C 180,E1 -16095.348,E2 -16095.348} C_VEL
LIN {X 0,Y 305.633,Z 203.226,A -85,B 0,C 180,E1 -16099.399,E2 -16099.399} C_VEL
LIN {X 0,Y 305.804,Z 203.202,A -85,B 0,C 180,E1 -16102.074,E2 -16102.074} C_VEL
LIN {X 0,Y 305.681,Z 203.221,A -85,B 0,C 180,E1 -16104.723,E2 -16104.723} C_VEL
LIN {X 0,Y 305.95,Z 203.188,A -85,B 0,C 180,E1 -16108.683,E2 -16108.683} C_VEL
LIN {X 0,Y 305.949,Z 203.185,A -85,B 0,C 180,E1 -16111.316,E2 -16111.316} C_VEL
LIN {X 0,Y 305.847,Z 203.202,A -85,B 0,C 180,E1 -16116.597,E2 -16116.597} C_VEL
LIN {X 0,Y 305.74,Z 203.21,A -85,B 0,C 180,E1 -16119.259,E2 -16119.259} C_VEL
LIN {X 0,Y 305.415,Z 203.251,A -85,B 0,C 180,E1 -16123.304,E2 -16123.304} C_VEL
LIN {X 0,Y 305.103,Z 203.466,A -85,B 0,C 180,E1 -16125.669,E2 -16125.669} C_VEL
LIN {X 0,Y 304.743,Z 207.184,A -85,B 0,C 180,E1 -16129.001,E2 -16129.001} C_VEL
LIN {X 0,Y 304.463,Z 211.885,A -85,B 0,C 180,E1 -16133.105,E2 -16133.105} C_VEL
LIN {X 0,Y 304.254,Z 215.318,A -85,B 0,C 180,E1 -16136.032,E2 -16136.032} C_VEL
LIN {X 0,Y 304.127,Z 218.728,A -85,B 0,C 180,E1 -16138.834,E2 -16138.834} C_VEL
LIN {X 0,Y 306.011,Z 229.908,A -85,B 0,C 180,E1 -16139.589,E2 -16139.589} C_VEL
LIN {X 0,Y 307.308,Z 239.024,A -85,B 0,C 180,E1 -16140.397,E2 -16140.397} C_VEL
LIN {X 0,Y 307.805,Z 243.954,A -85,B 0,C 180,E1 -16140.913,E2 -16140.913} C_VEL
LIN {X 0,Y 307.155,Z 252.449,A -85,B 0,C 180,E1 -16141.928,E2 -16141.928} C_VEL
LIN {X 0,Y 306.505,Z 260.111,A -85,B 0,C 180,E1 -16143.062,E2 -16143.062} C_VEL
LIN {X 0,Y 305.675,Z 268.497,A -85,B 0,C 180,E1 -16144.605,E2 -16144.605} C_VEL
LIN {X 0,Y 305.061,Z 275.389,A -85,B 0,C 180,E1 -16146.264,E2 -16146.264} C_VEL
LIN {X 0,Y 304.63,Z 279.751,A -85,B 0,C 180,E1 -16147.55,E2 -16147.55} C_VEL
LIN {X 0,Y 304.318,Z 282.73,A -85,B 0,C 180,E1 -16148.575,E2 -16148.575} C_VEL
LIN {X 0,Y 303.913,Z 286.714,A -85,B 0,C 180,E1 -16150.353,E2 -16150.353} C_VEL
LIN {X 0,Y 303.674,Z 289.685,A -85,B 0,C 180,E1 -16152.221,E2 -16152.221} C_VEL
LIN {X 0,Y 303.548,Z 291.582,A -85,B 0,C 180,E1 -16154.134,E2 -16154.134} C_VEL
LIN {X 0,Y 303.579,Z 292.365,A -85,B 0,C 180,E1 -16156.014,E2 -16156.014} C_VEL
LIN {X 0,Y 303.783,Z 292.057,A -85,B 0,C 180,E1 -16157.864,E2 -16157.864} C_VEL
LIN {X 0,Y 304.184,Z 290.673,A -85,B 0,C 180,E1 -16159.692,E2 -16159.692} C_VEL
LIN {X 0,Y 304.722,Z 288.017,A -85,B 0,C 180,E1 -16161.643,E2 -16161.643} C_VEL
LIN {X 0,Y 305.347,Z 284.871,A -85,B 0,C 180,E1 -16163.245,E2 -16163.245} C_VEL
LIN {X 0,Y 306.355,Z 279.234,A -85,B 0,C 180,E1 -16165.361,E2 -16165.361} C_VEL
LIN {X 0,Y 307.379,Z 273.432,A -85,B 0,C 180,E1 -16166.964,E2 -16166.964} C_VEL
LIN {X 0,Y 308.401,Z 266.973,A -85,B 0,C 180,E1 -16168.392,E2 -16168.392} C_VEL
LIN {X 0,Y 309.531,Z 260.018,A -85,B 0,C 180,E1 -16169.632,E2 -16169.632} C_VEL
LIN {X 0,Y 310.638,Z 251.328,A -85,B 0,C 180,E1 -16170.896,E2 -16170.896} C_VEL
LIN {X 0,Y 310.709,Z 246.823,A -85,B 0,C 180,E1 -16171.458,E2 -16171.458} C_VEL
LIN {X 0,Y 309.538,Z 239.009,A -85,B 0,C 180,E1 -16172.408,E2 -16172.408} C_VEL
LIN {X 0,Y 307.549,Z 230.002,A -85,B 0,C 180,E1 -16173.356,E2 -16173.356} C_VEL
LIN {X 0,Y 304.727,Z 220.13,A -85,B 0,C 180,E1 -16174.267,E2 -16174.267} C_VEL
LIN {X 0,Y 305.091,Z 215.903,A -85,B 0,C 180,E1 -16178.374,E2 -16178.374} C_VEL
LIN {X 0,Y 305.448,Z 213.075,A -85,B 0,C 180,E1 -16181.21,E2 -16181.21} C_VEL
LIN {X 0,Y 305.883,Z 209.115,A -85,B 0,C 180,E1 -16185.362,E2 -16185.362} C_VEL
LIN {X 0,Y 305.978,Z 206.704,A -85,B 0,C 180,E1 -16188.071,E2 -16188.071} C_VEL
LIN {X 0,Y 305.847,Z 203.681,A -85,B 0,C 180,E1 -16191.698,E2 -16191.698} C_VEL
LIN {X 0,Y 305.157,Z 203.327,A -85,B 0,C 180,E1 -16192.787,E2 -16192.787} C_VEL
LIN {X 0,Y 302.309,Z 203.648,A -85,B 0,C 180,E1 -16194.573,E2 -16194.573} C_VEL
LIN {X 0,Y 299.918,Z 203.973,A -85,B 0,C 180,E1 -16196.025,E2 -16196.025} C_VEL
LIN {X 0,Y 298.912,Z 204.07,A -85,B 0,C 180,E1 -16197.15,E2 -16197.15} C_VEL
LIN {X 0,Y 298.84,Z 204.074,A -85,B 0,C 180,E1 -16197.531,E2 -16197.531} C_VEL
LIN {X 0,Y 299.026,Z 204.051,A -85,B 0,C 180,E1 -16200.001,E2 -16200.001} C_VEL
LIN {X 0,Y 298.837,Z 204.073,A -85,B 0,C 180,E1 -16202.697,E2 -16202.697} C_VEL
LIN {X 0,Y 298.778,Z 204.082,A -85,B 0,C 180,E1 -16206.755,E2 -16206.755} C_VEL
LIN {X 0,Y 298.627,Z 204.102,A -85,B 0,C 180,E1 -16209.483,E2 -16209.483} C_VEL
LIN {X 0,Y 298.554,Z 204.11,A -85,B 0,C 180,E1 -16213.616,E2 -16213.616} C_VEL
LIN {X 0,Y 298.551,Z 204.11,A -85,B 0,C 180,E1 -16216.41,E2 -16216.41} C_VEL
LIN {X 0,Y 298.515,Z 204.115,A -85,B 0,C 180,E1 -16219.656,E2 -16219.656} C_VEL
LIN {X 0,Y 298.46,Z 204.121,A -85,B 0,C 180,E1 -16223.598,E2 -16223.598} C_VEL
LIN {X 0,Y 298.492,Z 204.117,A -85,B 0,C 180,E1 -16226.575,E2 -16226.575} C_VEL
LIN {X 0,Y 298.423,Z 204.126,A -85,B 0,C 180,E1 -16229.642,E2 -16229.642} C_VEL
LIN {X 0,Y 298.398,Z 204.127,A -85,B 0,C 180,E1 -16232.801,E2 -16232.801} C_VEL
LIN {X 0,Y 298.449,Z 204.123,A -85,B 0,C 180,E1 -16236.808,E2 -16236.808} C_VEL
LIN {X 0,Y 298.411,Z 204.129,A -85,B 0,C 180,E1 -16239.487,E2 -16239.487} C_VEL
LIN {X 0,Y 298.399,Z 204.214,A -85,B 0,C 180,E1 -16243.777,E2 -16243.777} C_VEL
LIN {X 0,Y 298.967,Z 207.35,A -85,B 0,C 180,E1 -16247.022,E2 -16247.022} C_VEL
LIN {X 0,Y 299.762,Z 211.366,A -85,B 0,C 180,E1 -16250.727,E2 -16250.727} C_VEL
LIN {X 0,Y 300.542,Z 215.613,A -85,B 0,C 180,E1 -16254.225,E2 -16254.225} C_VEL
LIN {X 0,Y 301.203,Z 220.021,A -85,B 0,C 180,E1 -16257.544,E2 -16257.544} C_VEL
LIN {X 0,Y 300.348,Z 224.577,A -85,B 0,C 180,E1 -16260.568,E2 -16260.568} C_VEL
LIN {X 0,Y 299.055,Z 231.584,A -85,B 0,C 180,E1 -16264.975,E2 -16264.975} C_VEL
LIN {X 0,Y 298.022,Z 238.815,A -85,B 0,C 180,E1 -16269.31,E2 -16269.31} C_VEL
LIN {X 0,Y 300.62,Z 251.459,A -85,B 0,C 180,E1 -16270.3,E2 -16270.3} C_VEL
LIN {X 0,Y 301.873,Z 260.421,A -85,B 0,C 180,E1 -16271.154,E2 -16271.154} C_VEL
LIN {X 0,Y 302.435,Z 268.681,A -85,B 0,C 180,E1 -16272.068,E2 -16272.068} C_VEL
LIN {X 0,Y 302.418,Z 277.527,A -85,B 0,C 180,E1 -16273.223,E2 -16273.223} C_VEL
LIN {X 0,Y 301.593,Z 284.572,A -85,B 0,C 180,E1 -16274.283,E2 -16274.283} C_VEL
LIN {X 0,Y 300.443,Z 291.082,A -85,B 0,C 180,E1 -16275.436,E2 -16275.436} C_VEL
LIN {X 0,Y 299.447,Z 297.293,A -85,B 0,C 180,E1 -16276.772,E2 -16276.772} C_VEL
LIN {X 0,Y 298.585,Z 302.469,A -85,B 0,C 180,E1 -16278.115,E2 -16278.115} C_VEL
LIN {X 0,Y 297.791,Z 307.771,A -85,B 0,C 180,E1 -16279.805,E2 -16279.805} C_VEL
LIN {X 0,Y 297.076,Z 312.729,A -85,B 0,C 180,E1 -16281.84,E2 -16281.84} C_VEL
LIN {X 0,Y 296.765,Z 315.161,A -85,B 0,C 180,E1 -16283.2,E2 -16283.2} C_VEL
LIN {X 0,Y 296.603,Z 317.039,A -85,B 0,C 180,E1 -16284.562,E2 -16284.562} C_VEL
LIN {X 0,Y 296.602,Z 318.411,A -85,B 0,C 180,E1 -16285.924,E2 -16285.924} C_VEL
LIN {X 0,Y 296.59,Z 319.294,A -85,B 0,C 180,E1 -16287.284,E2 -16287.284} C_VEL
LIN {X 0,Y 296.597,Z 319.661,A -85,B 0,C 180,E1 -16288.642,E2 -16288.642} C_VEL
LIN {X 0,Y 296.674,Z 319.434,A -85,B 0,C 180,E1 -16290,E2 -16290} C_VEL
LIN {X 0,Y 296.632,Z 318.698,A -85,B 0,C 180,E1 -16291.358,E2 -16291.358} C_VEL
LIN {X 0,Y 296.617,Z 317.464,A -85,B 0,C 180,E1 -16292.716,E2 -16292.716} C_VEL
LIN {X 0,Y 296.658,Z 314.557,A -85,B 0,C 180,E1 -16294.757,E2 -16294.757} C_VEL
LIN {X 0,Y 296.796,Z 310.338,A -85,B 0,C 180,E1 -16296.8,E2 -16296.8} C_VEL
LIN {X 0,Y 297.191,Z 304.429,A -85,B 0,C 180,E1 -16298.842,E2 -16298.842} C_VEL
LIN {X 0,Y 297.556,Z 299.485,A -85,B 0,C 180,E1 -16300.204,E2 -16300.204} C_VEL
LIN {X 0,Y 298.134,Z 293.516,A -85,B 0,C 180,E1 -16301.559,E2 -16301.559} C_VEL
LIN {X 0,Y 298.811,Z 286.234,A -85,B 0,C 180,E1 -16302.911,E2 -16302.911} C_VEL
LIN {X 0,Y 299.556,Z 278.451,A -85,B 0,C 180,E1 -16304.088,E2 -16304.088} C_VEL
LIN {X 0,Y 299.866,Z 273.182,A -85,B 0,C 180,E1 -16304.767,E2 -16304.767} C_VEL
LIN {X 0,Y 299.383,Z 264.216,A -85,B 0,C 180,E1 -16305.744,E2 -16305.744} C_VEL
LIN {X 0,Y 298.723,Z 255.74,A -85,B 0,C 180,E1 -16306.487,E2 -16306.487} C_VEL
LIN {X 0,Y 297.836,Z 245.813,A -85,B 0,C 180,E1 -16307.156,E2 -16307.156} C_VEL
LIN {X 0,Y 297.258,Z 240.255,A -85,B 0,C 180,E1 -16307.456,E2 -16307.456} C_VEL
LIN {X 0,Y 297.864,Z 233.242,A -85,B 0,C 180,E1 -16311.452,E2 -16311.452} C_VEL
LIN {X 0,Y 298.791,Z 225.717,A -85,B 0,C 180,E1 -16315.795,E2 -16315.795} C_VEL
LIN {X 0,Y 299.816,Z 218.837,A -85,B 0,C 180,E1 -16319.85,E2 -16319.85} C_VEL
LIN {X 0,Y 300.317,Z 215.614,A -85,B 0,C 180,E1 -16321.773,E2 -16321.773} C_VEL
LIN {X 0,Y 299.856,Z 211.743,A -85,B 0,C 180,E1 -16324.23,E2 -16324.23} C_VEL
LIN {X 0,Y 298.944,Z 206.529,A -85,B 0,C 180,E1 -16327.68,E2 -16327.68} C_VEL
LIN {X 0,Y 298.467,Z 204.125,A -85,B 0,C 180,E1 -16329.477,E2 -16329.477} C_VEL
LIN {X 0,Y 298.403,Z 204.125,A -85,B 0,C 180,E1 -16333.103,E2 -16333.103} C_VEL
LIN {X 0,Y 298.378,Z 204.128,A -85,B 0,C 180,E1 -16336.915,E2 -16336.915} C_VEL
LIN {X 0,Y 298.394,Z 204.126,A -85,B 0,C 180,E1 -16341.009,E2 -16341.009} C_VEL
LIN {X 0,Y 298.41,Z 204.126,A -85,B 0,C 180,E1 -16343.928,E2 -16343.928} C_VEL
LIN {X 0,Y 298.399,Z 204.125,A -85,B 0,C 180,E1 -16347.199,E2 -16347.199} C_VEL
LIN {X 0,Y 298.431,Z 204.121,A -85,B 0,C 180,E1 -16350.616,E2 -16350.616} C_VEL
LIN {X 0,Y 298.487,Z 204.115,A -85,B 0,C 180,E1 -16353.474,E2 -16353.474} C_VEL
LIN {X 0,Y 298.435,Z 204.12,A -85,B 0,C 180,E1 -16356.699,E2 -16356.699} C_VEL
LIN {X 0,Y 298.53,Z 204.108,A -85,B 0,C 180,E1 -16360.755,E2 -16360.755} C_VEL
LIN {X 0,Y 298.598,Z 204.101,A -85,B 0,C 180,E1 -16364.994,E2 -16364.994} C_VEL
LIN {X 0,Y 298.587,Z 204.103,A -85,B 0,C 180,E1 -16369.145,E2 -16369.145} C_VEL
LIN {X 0,Y 298.721,Z 204.086,A -85,B 0,C 180,E1 -16371.884,E2 -16371.884} C_VEL
LIN {X 0,Y 298.657,Z 204.093,A -85,B 0,C 180,E1 -16374.598,E2 -16374.598} C_VEL
LIN {X 0,Y 298.925,Z 204.059,A -85,B 0,C 180,E1 -16378.652,E2 -16378.652} C_VEL
LIN {X 0,Y 298.924,Z 204.063,A -85,B 0,C 180,E1 -16381.346,E2 -16381.346} C_VEL
LIN {X 0,Y 298.778,Z 204.08,A -85,B 0,C 180,E1 -16386.753,E2 -16386.753} C_VEL
LIN {X 0,Y 298.627,Z 204.097,A -85,B 0,C 180,E1 -16389.481,E2 -16389.481} C_VEL
LIN {X 0,Y 298.547,Z 204.106,A -85,B 0,C 180,E1 -16393.614,E2 -16393.614} C_VEL
LIN {X 0,Y 298.485,Z 204.116,A -85,B 0,C 180,E1 -16396.411,E2 -16396.411} C_VEL
LIN {X 0,Y 298.46,Z 204.117,A -85,B 0,C 180,E1 -16399.625,E2 -16399.625} C_VEL
LIN {X 0,Y 298.428,Z 204.12,A -85,B 0,C 180,E1 -16403.599,E2 -16403.599} C_VEL
LIN {X 0,Y 298.489,Z 204.118,A -85,B 0,C 180,E1 -16406.573,E2 -16406.573} C_VEL
LIN {X 0,Y 298.42,Z 204.122,A -85,B 0,C 180,E1 -16409.639,E2 -16409.639} C_VEL
LIN {X 0,Y 298.394,Z 204.126,A -85,B 0,C 180,E1 -16412.799,E2 -16412.799} C_VEL
LIN {X 0,Y 298.462,Z 204.118,A -85,B 0,C 180,E1 -16416.811,E2 -16416.811} C_VEL
LIN {X 0,Y 298.383,Z 204.126,A -85,B 0,C 180,E1 -16421.086,E2 -16421.086} C_VEL
LIN {X 0,Y 298.395,Z 204.125,A -85,B 0,C 180,E1 -16423.102,E2 -16423.102} C_VEL
LIN {X 0,Y 298.398,Z 204.125,A -85,B 0,C 180,E1 -16426.919,E2 -16426.919} C_VEL
LIN {X 0,Y 298.41,Z 204.124,A -85,B 0,C 180,E1 -16431.002,E2 -16431.002} C_VEL
LIN {X 0,Y 298.413,Z 204.126,A -85,B 0,C 180,E1 -16433.929,E2 -16433.929} C_VEL
LIN {X 0,Y 298.39,Z 204.128,A -85,B 0,C 180,E1 -16437.982,E2 -16437.982} C_VEL
LIN {X 0,Y 298.469,Z 204.118,A -85,B 0,C 180,E1 -16441.904,E2 -16441.904} C_VEL
LIN {X 0,Y 298.479,Z 204.116,A -85,B 0,C 180,E1 -16444.923,E2 -16444.923} C_VEL
LIN {X 0,Y 298.443,Z 204.125,A -85,B 0,C 180,E1 -16449.314,E2 -16449.314} C_VEL
LIN {X 0,Y 298.531,Z 204.108,A -85,B 0,C 180,E1 -16452.179,E2 -16452.179} C_VEL
LIN {X 0,Y 298.586,Z 204.105,A -85,B 0,C 180,E1 -16454.994,E2 -16454.994} C_VEL
LIN {X 0,Y 298.588,Z 204.105,A -85,B 0,C 180,E1 -16459.146,E2 -16459.146} C_VEL
LIN {X 0,Y 298.75,Z 204.08,A -85,B 0,C 180,E1 -16461.885,E2 -16461.885} C_VEL
LIN {X 0,Y 298.652,Z 204.096,A -85,B 0,C 180,E1 -16464.599,E2 -16464.599} C_VEL
LIN {X 0,Y 298.917,Z 204.064,A -85,B 0,C 180,E1 -16468.653,E2 -16468.653} C_VEL
LIN {X 0,Y 298.915,Z 204.061,A -85,B 0,C 180,E1 -16471.347,E2 -16471.347} C_VEL
LIN {X 0,Y 298.794,Z 204.079,A -85,B 0,C 180,E1 -16476.754,E2 -16476.754} C_VEL
LIN {X 0,Y 298.675,Z 204.09,A -85,B 0,C 180,E1 -16479.48,E2 -16479.48} C_VEL
LIN {X 0,Y 298.348,Z 204.132,A -85,B 0,C 180,E1 -16483.625,E2 -16483.625} C_VEL
LIN {X 0,Y 298.064,Z 204.195,A -85,B 0,C 180,E1 -16485.558,E2 -16485.558} C_VEL
LIN {X 0,Y 297.653,Z 208.309,A -85,B 0,C 180,E1 -16489.303,E2 -16489.303} C_VEL
